   AxisStore[14].Axis[12].Pos13.Position := 0.0;
   AxisStore[14].Axis[12].Pos13.Speed := 0;
   AxisStore[14].Axis[12].Pos13.Reached := FALSE;
   AxisStore[14].Axis[12].Pos14.Position := 0.0;
   AxisStore[14].Axis[12].Pos14.Speed := 0;
   AxisStore[14].Axis[12].Pos14.Reached := FALSE;
   AxisStore[14].Axis[12].Pos15.Position := 0.0;
   AxisStore[14].Axis[12].Pos15.Speed := 0;
   AxisStore[14].Axis[12].Pos15.Reached := FALSE;
   AxisStore[14].Axis[12].Pos16.Position := 0.0;
   AxisStore[14].Axis[12].Pos16.Speed := 0;
   AxisStore[14].Axis[12].Pos16.Reached := FALSE;
   AxisStore[14].Axis[12].Pos17.Position := 0.0;
   AxisStore[14].Axis[12].Pos17.Speed := 0;
   AxisStore[14].Axis[12].Pos17.Reached := FALSE;
   AxisStore[14].Axis[12].Pos18.Position := 0.0;
   AxisStore[14].Axis[12].Pos18.Speed := 0;
   AxisStore[14].Axis[12].Pos18.Reached := FALSE;
   AxisStore[14].Axis[12].Pos19.Position := 0.0;
   AxisStore[14].Axis[12].Pos19.Speed := 0;
   AxisStore[14].Axis[12].Pos19.Reached := FALSE;
   AxisStore[14].Axis[12].Pos20.Position := 0.0;
   AxisStore[14].Axis[12].Pos20.Speed := 0;
   AxisStore[14].Axis[12].Pos20.Reached := FALSE;
   AxisStore[14].Axis[12].Pos21.Position := 0.0;
   AxisStore[14].Axis[12].Pos21.Speed := 0;
   AxisStore[14].Axis[12].Pos21.Reached := FALSE;
   AxisStore[14].Axis[12].Pos22.Position := 0.0;
   AxisStore[14].Axis[12].Pos22.Speed := 0;
   AxisStore[14].Axis[12].Pos22.Reached := FALSE;
   AxisStore[14].Axis[12].Pos23.Position := 0.0;
   AxisStore[14].Axis[12].Pos23.Speed := 0;
   AxisStore[14].Axis[12].Pos23.Reached := FALSE;
   AxisStore[14].Axis[12].Pos24.Position := 0.0;
   AxisStore[14].Axis[12].Pos24.Speed := 0;
   AxisStore[14].Axis[12].Pos24.Reached := FALSE;
   AxisStore[14].Axis[12].Pos25.Position := 0.0;
   AxisStore[14].Axis[12].Pos25.Speed := 0;
   AxisStore[14].Axis[12].Pos25.Reached := FALSE;
   AxisStore[14].Axis[12].Pos26.Position := 0.0;
   AxisStore[14].Axis[12].Pos26.Speed := 0;
   AxisStore[14].Axis[12].Pos26.Reached := FALSE;
   AxisStore[14].Axis[12].Pos27.Position := 0.0;
   AxisStore[14].Axis[12].Pos27.Speed := 0;
   AxisStore[14].Axis[12].Pos27.Reached := FALSE;
   AxisStore[14].Axis[12].Pos28.Position := 0.0;
   AxisStore[14].Axis[12].Pos28.Speed := 0;
   AxisStore[14].Axis[12].Pos28.Reached := FALSE;
   AxisStore[14].Axis[12].Pos29.Position := 0.0;
   AxisStore[14].Axis[12].Pos29.Speed := 0;
   AxisStore[14].Axis[12].Pos29.Reached := FALSE;
   AxisStore[14].Axis[12].Pos30.Position := 0.0;
   AxisStore[14].Axis[12].Pos30.Speed := 0;
   AxisStore[14].Axis[12].Pos30.Reached := FALSE;
   AxisStore[14].Axis[13].Pos1.Position := 0.0;
   AxisStore[14].Axis[13].Pos1.Speed := 0;
   AxisStore[14].Axis[13].Pos1.Reached := FALSE;
   AxisStore[14].Axis[13].Pos2.Position := 0.0;
   AxisStore[14].Axis[13].Pos2.Speed := 0;
   AxisStore[14].Axis[13].Pos2.Reached := FALSE;
   AxisStore[14].Axis[13].Pos3.Position := 0.0;
   AxisStore[14].Axis[13].Pos3.Speed := 0;
   AxisStore[14].Axis[13].Pos3.Reached := FALSE;
   AxisStore[14].Axis[13].Pos4.Position := 0.0;
   AxisStore[14].Axis[13].Pos4.Speed := 0;
   AxisStore[14].Axis[13].Pos4.Reached := FALSE;
   AxisStore[14].Axis[13].Pos5.Position := 0.0;
   AxisStore[14].Axis[13].Pos5.Speed := 0;
   AxisStore[14].Axis[13].Pos5.Reached := FALSE;
   AxisStore[14].Axis[13].Pos6.Position := 0.0;
   AxisStore[14].Axis[13].Pos6.Speed := 0;
   AxisStore[14].Axis[13].Pos6.Reached := FALSE;
   AxisStore[14].Axis[13].Pos7.Position := 0.0;
   AxisStore[14].Axis[13].Pos7.Speed := 0;
   AxisStore[14].Axis[13].Pos7.Reached := FALSE;
   AxisStore[14].Axis[13].Pos8.Position := 0.0;
   AxisStore[14].Axis[13].Pos8.Speed := 0;
   AxisStore[14].Axis[13].Pos8.Reached := FALSE;
   AxisStore[14].Axis[13].Pos9.Position := 0.0;
   AxisStore[14].Axis[13].Pos9.Speed := 0;
   AxisStore[14].Axis[13].Pos9.Reached := FALSE;
   AxisStore[14].Axis[13].Pos10.Position := 0.0;
   AxisStore[14].Axis[13].Pos10.Speed := 0;
   AxisStore[14].Axis[13].Pos10.Reached := FALSE;
   AxisStore[14].Axis[13].Pos11.Position := 0.0;
   AxisStore[14].Axis[13].Pos11.Speed := 0;
   AxisStore[14].Axis[13].Pos11.Reached := FALSE;
   AxisStore[14].Axis[13].Pos12.Position := 0.0;
   AxisStore[14].Axis[13].Pos12.Speed := 0;
   AxisStore[14].Axis[13].Pos12.Reached := FALSE;
   AxisStore[14].Axis[13].Pos13.Position := 0.0;
   AxisStore[14].Axis[13].Pos13.Speed := 0;
   AxisStore[14].Axis[13].Pos13.Reached := FALSE;
   AxisStore[14].Axis[13].Pos14.Position := 0.0;
   AxisStore[14].Axis[13].Pos14.Speed := 0;
   AxisStore[14].Axis[13].Pos14.Reached := FALSE;
   AxisStore[14].Axis[13].Pos15.Position := 0.0;
   AxisStore[14].Axis[13].Pos15.Speed := 0;
   AxisStore[14].Axis[13].Pos15.Reached := FALSE;
   AxisStore[14].Axis[13].Pos16.Position := 0.0;
   AxisStore[14].Axis[13].Pos16.Speed := 0;
   AxisStore[14].Axis[13].Pos16.Reached := FALSE;
   AxisStore[14].Axis[13].Pos17.Position := 0.0;
   AxisStore[14].Axis[13].Pos17.Speed := 0;
   AxisStore[14].Axis[13].Pos17.Reached := FALSE;
   AxisStore[14].Axis[13].Pos18.Position := 0.0;
   AxisStore[14].Axis[13].Pos18.Speed := 0;
   AxisStore[14].Axis[13].Pos18.Reached := FALSE;
   AxisStore[14].Axis[13].Pos19.Position := 0.0;
   AxisStore[14].Axis[13].Pos19.Speed := 0;
   AxisStore[14].Axis[13].Pos19.Reached := FALSE;
   AxisStore[14].Axis[13].Pos20.Position := 0.0;
   AxisStore[14].Axis[13].Pos20.Speed := 0;
   AxisStore[14].Axis[13].Pos20.Reached := FALSE;
   AxisStore[14].Axis[13].Pos21.Position := 0.0;
   AxisStore[14].Axis[13].Pos21.Speed := 0;
   AxisStore[14].Axis[13].Pos21.Reached := FALSE;
   AxisStore[14].Axis[13].Pos22.Position := 0.0;
   AxisStore[14].Axis[13].Pos22.Speed := 0;
   AxisStore[14].Axis[13].Pos22.Reached := FALSE;
   AxisStore[14].Axis[13].Pos23.Position := 0.0;
   AxisStore[14].Axis[13].Pos23.Speed := 0;
   AxisStore[14].Axis[13].Pos23.Reached := FALSE;
   AxisStore[14].Axis[13].Pos24.Position := 0.0;
   AxisStore[14].Axis[13].Pos24.Speed := 0;
   AxisStore[14].Axis[13].Pos24.Reached := FALSE;
   AxisStore[14].Axis[13].Pos25.Position := 0.0;
   AxisStore[14].Axis[13].Pos25.Speed := 0;
   AxisStore[14].Axis[13].Pos25.Reached := FALSE;
   AxisStore[14].Axis[13].Pos26.Position := 0.0;
   AxisStore[14].Axis[13].Pos26.Speed := 0;
   AxisStore[14].Axis[13].Pos26.Reached := FALSE;
   AxisStore[14].Axis[13].Pos27.Position := 0.0;
   AxisStore[14].Axis[13].Pos27.Speed := 0;
   AxisStore[14].Axis[13].Pos27.Reached := FALSE;
   AxisStore[14].Axis[13].Pos28.Position := 0.0;
   AxisStore[14].Axis[13].Pos28.Speed := 0;
   AxisStore[14].Axis[13].Pos28.Reached := FALSE;
   AxisStore[14].Axis[13].Pos29.Position := 0.0;
   AxisStore[14].Axis[13].Pos29.Speed := 0;
   AxisStore[14].Axis[13].Pos29.Reached := FALSE;
   AxisStore[14].Axis[13].Pos30.Position := 0.0;
   AxisStore[14].Axis[13].Pos30.Speed := 0;
   AxisStore[14].Axis[13].Pos30.Reached := FALSE;
   AxisStore[14].Axis[14].Pos1.Position := 0.0;
   AxisStore[14].Axis[14].Pos1.Speed := 0;
   AxisStore[14].Axis[14].Pos1.Reached := FALSE;
   AxisStore[14].Axis[14].Pos2.Position := 0.0;
   AxisStore[14].Axis[14].Pos2.Speed := 0;
   AxisStore[14].Axis[14].Pos2.Reached := FALSE;
   AxisStore[14].Axis[14].Pos3.Position := 0.0;
   AxisStore[14].Axis[14].Pos3.Speed := 0;
   AxisStore[14].Axis[14].Pos3.Reached := FALSE;
   AxisStore[14].Axis[14].Pos4.Position := 0.0;
   AxisStore[14].Axis[14].Pos4.Speed := 0;
   AxisStore[14].Axis[14].Pos4.Reached := FALSE;
   AxisStore[14].Axis[14].Pos5.Position := 0.0;
   AxisStore[14].Axis[14].Pos5.Speed := 0;
   AxisStore[14].Axis[14].Pos5.Reached := FALSE;
   AxisStore[14].Axis[14].Pos6.Position := 0.0;
   AxisStore[14].Axis[14].Pos6.Speed := 0;
   AxisStore[14].Axis[14].Pos6.Reached := FALSE;
   AxisStore[14].Axis[14].Pos7.Position := 0.0;
   AxisStore[14].Axis[14].Pos7.Speed := 0;
   AxisStore[14].Axis[14].Pos7.Reached := FALSE;
   AxisStore[14].Axis[14].Pos8.Position := 0.0;
   AxisStore[14].Axis[14].Pos8.Speed := 0;
   AxisStore[14].Axis[14].Pos8.Reached := FALSE;
   AxisStore[14].Axis[14].Pos9.Position := 0.0;
   AxisStore[14].Axis[14].Pos9.Speed := 0;
   AxisStore[14].Axis[14].Pos9.Reached := FALSE;
   AxisStore[14].Axis[14].Pos10.Position := 0.0;
   AxisStore[14].Axis[14].Pos10.Speed := 0;
   AxisStore[14].Axis[14].Pos10.Reached := FALSE;
   AxisStore[14].Axis[14].Pos11.Position := 0.0;
   AxisStore[14].Axis[14].Pos11.Speed := 0;
   AxisStore[14].Axis[14].Pos11.Reached := FALSE;
   AxisStore[14].Axis[14].Pos12.Position := 0.0;
   AxisStore[14].Axis[14].Pos12.Speed := 0;
   AxisStore[14].Axis[14].Pos12.Reached := FALSE;
   AxisStore[14].Axis[14].Pos13.Position := 0.0;
   AxisStore[14].Axis[14].Pos13.Speed := 0;
   AxisStore[14].Axis[14].Pos13.Reached := FALSE;
   AxisStore[14].Axis[14].Pos14.Position := 0.0;
   AxisStore[14].Axis[14].Pos14.Speed := 0;
   AxisStore[14].Axis[14].Pos14.Reached := FALSE;
   AxisStore[14].Axis[14].Pos15.Position := 0.0;
   AxisStore[14].Axis[14].Pos15.Speed := 0;
   AxisStore[14].Axis[14].Pos15.Reached := FALSE;
   AxisStore[14].Axis[14].Pos16.Position := 0.0;
   AxisStore[14].Axis[14].Pos16.Speed := 0;
   AxisStore[14].Axis[14].Pos16.Reached := FALSE;
   AxisStore[14].Axis[14].Pos17.Position := 0.0;
   AxisStore[14].Axis[14].Pos17.Speed := 0;
   AxisStore[14].Axis[14].Pos17.Reached := FALSE;
   AxisStore[14].Axis[14].Pos18.Position := 0.0;
   AxisStore[14].Axis[14].Pos18.Speed := 0;
   AxisStore[14].Axis[14].Pos18.Reached := FALSE;
   AxisStore[14].Axis[14].Pos19.Position := 0.0;
   AxisStore[14].Axis[14].Pos19.Speed := 0;
   AxisStore[14].Axis[14].Pos19.Reached := FALSE;
   AxisStore[14].Axis[14].Pos20.Position := 0.0;
   AxisStore[14].Axis[14].Pos20.Speed := 0;
   AxisStore[14].Axis[14].Pos20.Reached := FALSE;
   AxisStore[14].Axis[14].Pos21.Position := 0.0;
   AxisStore[14].Axis[14].Pos21.Speed := 0;
   AxisStore[14].Axis[14].Pos21.Reached := FALSE;
   AxisStore[14].Axis[14].Pos22.Position := 0.0;
   AxisStore[14].Axis[14].Pos22.Speed := 0;
   AxisStore[14].Axis[14].Pos22.Reached := FALSE;
   AxisStore[14].Axis[14].Pos23.Position := 0.0;
   AxisStore[14].Axis[14].Pos23.Speed := 0;
   AxisStore[14].Axis[14].Pos23.Reached := FALSE;
   AxisStore[14].Axis[14].Pos24.Position := 0.0;
   AxisStore[14].Axis[14].Pos24.Speed := 0;
   AxisStore[14].Axis[14].Pos24.Reached := FALSE;
   AxisStore[14].Axis[14].Pos25.Position := 0.0;
   AxisStore[14].Axis[14].Pos25.Speed := 0;
   AxisStore[14].Axis[14].Pos25.Reached := FALSE;
   AxisStore[14].Axis[14].Pos26.Position := 0.0;
   AxisStore[14].Axis[14].Pos26.Speed := 0;
   AxisStore[14].Axis[14].Pos26.Reached := FALSE;
   AxisStore[14].Axis[14].Pos27.Position := 0.0;
   AxisStore[14].Axis[14].Pos27.Speed := 0;
   AxisStore[14].Axis[14].Pos27.Reached := FALSE;
   AxisStore[14].Axis[14].Pos28.Position := 0.0;
   AxisStore[14].Axis[14].Pos28.Speed := 0;
   AxisStore[14].Axis[14].Pos28.Reached := FALSE;
   AxisStore[14].Axis[14].Pos29.Position := 0.0;
   AxisStore[14].Axis[14].Pos29.Speed := 0;
   AxisStore[14].Axis[14].Pos29.Reached := FALSE;
   AxisStore[14].Axis[14].Pos30.Position := 0.0;
   AxisStore[14].Axis[14].Pos30.Speed := 0;
   AxisStore[14].Axis[14].Pos30.Reached := FALSE;
   AxisStore[14].Axis[15].Pos1.Position := 0.0;
   AxisStore[14].Axis[15].Pos1.Speed := 0;
   AxisStore[14].Axis[15].Pos1.Reached := FALSE;
   AxisStore[14].Axis[15].Pos2.Position := 0.0;
   AxisStore[14].Axis[15].Pos2.Speed := 0;
   AxisStore[14].Axis[15].Pos2.Reached := FALSE;
   AxisStore[14].Axis[15].Pos3.Position := 0.0;
   AxisStore[14].Axis[15].Pos3.Speed := 0;
   AxisStore[14].Axis[15].Pos3.Reached := FALSE;
   AxisStore[14].Axis[15].Pos4.Position := 0.0;
   AxisStore[14].Axis[15].Pos4.Speed := 0;
   AxisStore[14].Axis[15].Pos4.Reached := FALSE;
   AxisStore[14].Axis[15].Pos5.Position := 0.0;
   AxisStore[14].Axis[15].Pos5.Speed := 0;
   AxisStore[14].Axis[15].Pos5.Reached := FALSE;
   AxisStore[14].Axis[15].Pos6.Position := 0.0;
   AxisStore[14].Axis[15].Pos6.Speed := 0;
   AxisStore[14].Axis[15].Pos6.Reached := FALSE;
   AxisStore[14].Axis[15].Pos7.Position := 0.0;
   AxisStore[14].Axis[15].Pos7.Speed := 0;
   AxisStore[14].Axis[15].Pos7.Reached := FALSE;
   AxisStore[14].Axis[15].Pos8.Position := 0.0;
   AxisStore[14].Axis[15].Pos8.Speed := 0;
   AxisStore[14].Axis[15].Pos8.Reached := FALSE;
   AxisStore[14].Axis[15].Pos9.Position := 0.0;
   AxisStore[14].Axis[15].Pos9.Speed := 0;
   AxisStore[14].Axis[15].Pos9.Reached := FALSE;
   AxisStore[14].Axis[15].Pos10.Position := 0.0;
   AxisStore[14].Axis[15].Pos10.Speed := 0;
   AxisStore[14].Axis[15].Pos10.Reached := FALSE;
   AxisStore[14].Axis[15].Pos11.Position := 0.0;
   AxisStore[14].Axis[15].Pos11.Speed := 0;
   AxisStore[14].Axis[15].Pos11.Reached := FALSE;
   AxisStore[14].Axis[15].Pos12.Position := 0.0;
   AxisStore[14].Axis[15].Pos12.Speed := 0;
   AxisStore[14].Axis[15].Pos12.Reached := FALSE;
   AxisStore[14].Axis[15].Pos13.Position := 0.0;
   AxisStore[14].Axis[15].Pos13.Speed := 0;
   AxisStore[14].Axis[15].Pos13.Reached := FALSE;
   AxisStore[14].Axis[15].Pos14.Position := 0.0;
   AxisStore[14].Axis[15].Pos14.Speed := 0;
   AxisStore[14].Axis[15].Pos14.Reached := FALSE;
   AxisStore[14].Axis[15].Pos15.Position := 0.0;
   AxisStore[14].Axis[15].Pos15.Speed := 0;
   AxisStore[14].Axis[15].Pos15.Reached := FALSE;
   AxisStore[14].Axis[15].Pos16.Position := 0.0;
   AxisStore[14].Axis[15].Pos16.Speed := 0;
   AxisStore[14].Axis[15].Pos16.Reached := FALSE;
   AxisStore[14].Axis[15].Pos17.Position := 0.0;
   AxisStore[14].Axis[15].Pos17.Speed := 0;
   AxisStore[14].Axis[15].Pos17.Reached := FALSE;
   AxisStore[14].Axis[15].Pos18.Position := 0.0;
   AxisStore[14].Axis[15].Pos18.Speed := 0;
   AxisStore[14].Axis[15].Pos18.Reached := FALSE;
   AxisStore[14].Axis[15].Pos19.Position := 0.0;
   AxisStore[14].Axis[15].Pos19.Speed := 0;
   AxisStore[14].Axis[15].Pos19.Reached := FALSE;
   AxisStore[14].Axis[15].Pos20.Position := 0.0;
   AxisStore[14].Axis[15].Pos20.Speed := 0;
   AxisStore[14].Axis[15].Pos20.Reached := FALSE;
   AxisStore[14].Axis[15].Pos21.Position := 0.0;
   AxisStore[14].Axis[15].Pos21.Speed := 0;
   AxisStore[14].Axis[15].Pos21.Reached := FALSE;
   AxisStore[14].Axis[15].Pos22.Position := 0.0;
   AxisStore[14].Axis[15].Pos22.Speed := 0;
   AxisStore[14].Axis[15].Pos22.Reached := FALSE;
   AxisStore[14].Axis[15].Pos23.Position := 0.0;
   AxisStore[14].Axis[15].Pos23.Speed := 0;
   AxisStore[14].Axis[15].Pos23.Reached := FALSE;
   AxisStore[14].Axis[15].Pos24.Position := 0.0;
   AxisStore[14].Axis[15].Pos24.Speed := 0;
   AxisStore[14].Axis[15].Pos24.Reached := FALSE;
   AxisStore[14].Axis[15].Pos25.Position := 0.0;
   AxisStore[14].Axis[15].Pos25.Speed := 0;
   AxisStore[14].Axis[15].Pos25.Reached := FALSE;
   AxisStore[14].Axis[15].Pos26.Position := 0.0;
   AxisStore[14].Axis[15].Pos26.Speed := 0;
   AxisStore[14].Axis[15].Pos26.Reached := FALSE;
   AxisStore[14].Axis[15].Pos27.Position := 0.0;
   AxisStore[14].Axis[15].Pos27.Speed := 0;
   AxisStore[14].Axis[15].Pos27.Reached := FALSE;
   AxisStore[14].Axis[15].Pos28.Position := 0.0;
   AxisStore[14].Axis[15].Pos28.Speed := 0;
   AxisStore[14].Axis[15].Pos28.Reached := FALSE;
   AxisStore[14].Axis[15].Pos29.Position := 0.0;
   AxisStore[14].Axis[15].Pos29.Speed := 0;
   AxisStore[14].Axis[15].Pos29.Reached := FALSE;
   AxisStore[14].Axis[15].Pos30.Position := 0.0;
   AxisStore[14].Axis[15].Pos30.Speed := 0;
   AxisStore[14].Axis[15].Pos30.Reached := FALSE;
   AxisStore[15].Axis[1].Pos1.Position := 0.0;
   AxisStore[15].Axis[1].Pos1.Speed := 0;
   AxisStore[15].Axis[1].Pos1.Reached := FALSE;
   AxisStore[15].Axis[1].Pos2.Position := 0.0;
   AxisStore[15].Axis[1].Pos2.Speed := 0;
   AxisStore[15].Axis[1].Pos2.Reached := FALSE;
   AxisStore[15].Axis[1].Pos3.Position := 0.0;
   AxisStore[15].Axis[1].Pos3.Speed := 0;
   AxisStore[15].Axis[1].Pos3.Reached := FALSE;
   AxisStore[15].Axis[1].Pos4.Position := 0.0;
   AxisStore[15].Axis[1].Pos4.Speed := 0;
   AxisStore[15].Axis[1].Pos4.Reached := FALSE;
   AxisStore[15].Axis[1].Pos5.Position := 0.0;
   AxisStore[15].Axis[1].Pos5.Speed := 0;
   AxisStore[15].Axis[1].Pos5.Reached := FALSE;
   AxisStore[15].Axis[1].Pos6.Position := 0.0;
   AxisStore[15].Axis[1].Pos6.Speed := 0;
   AxisStore[15].Axis[1].Pos6.Reached := FALSE;
   AxisStore[15].Axis[1].Pos7.Position := 0.0;
   AxisStore[15].Axis[1].Pos7.Speed := 0;
   AxisStore[15].Axis[1].Pos7.Reached := FALSE;
   AxisStore[15].Axis[1].Pos8.Position := 0.0;
   AxisStore[15].Axis[1].Pos8.Speed := 0;
   AxisStore[15].Axis[1].Pos8.Reached := FALSE;
   AxisStore[15].Axis[1].Pos9.Position := 0.0;
   AxisStore[15].Axis[1].Pos9.Speed := 0;
   AxisStore[15].Axis[1].Pos9.Reached := FALSE;
   AxisStore[15].Axis[1].Pos10.Position := 0.0;
   AxisStore[15].Axis[1].Pos10.Speed := 0;
   AxisStore[15].Axis[1].Pos10.Reached := FALSE;
   AxisStore[15].Axis[1].Pos11.Position := 0.0;
   AxisStore[15].Axis[1].Pos11.Speed := 0;
   AxisStore[15].Axis[1].Pos11.Reached := FALSE;
   AxisStore[15].Axis[1].Pos12.Position := 0.0;
   AxisStore[15].Axis[1].Pos12.Speed := 0;
   AxisStore[15].Axis[1].Pos12.Reached := FALSE;
   AxisStore[15].Axis[1].Pos13.Position := 0.0;
   AxisStore[15].Axis[1].Pos13.Speed := 0;
   AxisStore[15].Axis[1].Pos13.Reached := FALSE;
   AxisStore[15].Axis[1].Pos14.Position := 0.0;
   AxisStore[15].Axis[1].Pos14.Speed := 0;
   AxisStore[15].Axis[1].Pos14.Reached := FALSE;
   AxisStore[15].Axis[1].Pos15.Position := 0.0;
   AxisStore[15].Axis[1].Pos15.Speed := 0;
   AxisStore[15].Axis[1].Pos15.Reached := FALSE;
   AxisStore[15].Axis[1].Pos16.Position := 0.0;
   AxisStore[15].Axis[1].Pos16.Speed := 0;
   AxisStore[15].Axis[1].Pos16.Reached := FALSE;
   AxisStore[15].Axis[1].Pos17.Position := 0.0;
   AxisStore[15].Axis[1].Pos17.Speed := 0;
   AxisStore[15].Axis[1].Pos17.Reached := FALSE;
   AxisStore[15].Axis[1].Pos18.Position := 0.0;
   AxisStore[15].Axis[1].Pos18.Speed := 0;
   AxisStore[15].Axis[1].Pos18.Reached := FALSE;
   AxisStore[15].Axis[1].Pos19.Position := 0.0;
   AxisStore[15].Axis[1].Pos19.Speed := 0;
   AxisStore[15].Axis[1].Pos19.Reached := FALSE;
   AxisStore[15].Axis[1].Pos20.Position := 0.0;
   AxisStore[15].Axis[1].Pos20.Speed := 0;
   AxisStore[15].Axis[1].Pos20.Reached := FALSE;
   AxisStore[15].Axis[1].Pos21.Position := 0.0;
   AxisStore[15].Axis[1].Pos21.Speed := 0;
   AxisStore[15].Axis[1].Pos21.Reached := FALSE;
   AxisStore[15].Axis[1].Pos22.Position := 0.0;
   AxisStore[15].Axis[1].Pos22.Speed := 0;
   AxisStore[15].Axis[1].Pos22.Reached := FALSE;
   AxisStore[15].Axis[1].Pos23.Position := 0.0;
   AxisStore[15].Axis[1].Pos23.Speed := 0;
   AxisStore[15].Axis[1].Pos23.Reached := FALSE;
   AxisStore[15].Axis[1].Pos24.Position := 0.0;
   AxisStore[15].Axis[1].Pos24.Speed := 0;
   AxisStore[15].Axis[1].Pos24.Reached := FALSE;
   AxisStore[15].Axis[1].Pos25.Position := 0.0;
   AxisStore[15].Axis[1].Pos25.Speed := 0;
   AxisStore[15].Axis[1].Pos25.Reached := FALSE;
   AxisStore[15].Axis[1].Pos26.Position := 0.0;
   AxisStore[15].Axis[1].Pos26.Speed := 0;
   AxisStore[15].Axis[1].Pos26.Reached := FALSE;
   AxisStore[15].Axis[1].Pos27.Position := 0.0;
   AxisStore[15].Axis[1].Pos27.Speed := 0;
   AxisStore[15].Axis[1].Pos27.Reached := FALSE;
   AxisStore[15].Axis[1].Pos28.Position := 0.0;
   AxisStore[15].Axis[1].Pos28.Speed := 0;
   AxisStore[15].Axis[1].Pos28.Reached := FALSE;
   AxisStore[15].Axis[1].Pos29.Position := 0.0;
   AxisStore[15].Axis[1].Pos29.Speed := 0;
   AxisStore[15].Axis[1].Pos29.Reached := FALSE;
   AxisStore[15].Axis[1].Pos30.Position := 0.0;
   AxisStore[15].Axis[1].Pos30.Speed := 0;
   AxisStore[15].Axis[1].Pos30.Reached := FALSE;
   AxisStore[15].Axis[2].Pos1.Position := 0.0;
   AxisStore[15].Axis[2].Pos1.Speed := 0;
   AxisStore[15].Axis[2].Pos1.Reached := FALSE;
   AxisStore[15].Axis[2].Pos2.Position := 0.0;
   AxisStore[15].Axis[2].Pos2.Speed := 0;
   AxisStore[15].Axis[2].Pos2.Reached := FALSE;
   AxisStore[15].Axis[2].Pos3.Position := 0.0;
   AxisStore[15].Axis[2].Pos3.Speed := 0;
   AxisStore[15].Axis[2].Pos3.Reached := FALSE;
   AxisStore[15].Axis[2].Pos4.Position := 0.0;
   AxisStore[15].Axis[2].Pos4.Speed := 0;
   AxisStore[15].Axis[2].Pos4.Reached := FALSE;
   AxisStore[15].Axis[2].Pos5.Position := 0.0;
   AxisStore[15].Axis[2].Pos5.Speed := 0;
   AxisStore[15].Axis[2].Pos5.Reached := FALSE;
   AxisStore[15].Axis[2].Pos6.Position := 0.0;
   AxisStore[15].Axis[2].Pos6.Speed := 0;
   AxisStore[15].Axis[2].Pos6.Reached := FALSE;
   AxisStore[15].Axis[2].Pos7.Position := 0.0;
   AxisStore[15].Axis[2].Pos7.Speed := 0;
   AxisStore[15].Axis[2].Pos7.Reached := FALSE;
   AxisStore[15].Axis[2].Pos8.Position := 0.0;
   AxisStore[15].Axis[2].Pos8.Speed := 0;
   AxisStore[15].Axis[2].Pos8.Reached := FALSE;
   AxisStore[15].Axis[2].Pos9.Position := 0.0;
   AxisStore[15].Axis[2].Pos9.Speed := 0;
   AxisStore[15].Axis[2].Pos9.Reached := FALSE;
   AxisStore[15].Axis[2].Pos10.Position := 0.0;
   AxisStore[15].Axis[2].Pos10.Speed := 0;
   AxisStore[15].Axis[2].Pos10.Reached := FALSE;
   AxisStore[15].Axis[2].Pos11.Position := 0.0;
   AxisStore[15].Axis[2].Pos11.Speed := 0;
   AxisStore[15].Axis[2].Pos11.Reached := FALSE;
   AxisStore[15].Axis[2].Pos12.Position := 0.0;
   AxisStore[15].Axis[2].Pos12.Speed := 0;
   AxisStore[15].Axis[2].Pos12.Reached := FALSE;
   AxisStore[15].Axis[2].Pos13.Position := 0.0;
   AxisStore[15].Axis[2].Pos13.Speed := 0;
   AxisStore[15].Axis[2].Pos13.Reached := FALSE;
   AxisStore[15].Axis[2].Pos14.Position := 0.0;
   AxisStore[15].Axis[2].Pos14.Speed := 0;
   AxisStore[15].Axis[2].Pos14.Reached := FALSE;
   AxisStore[15].Axis[2].Pos15.Position := 0.0;
   AxisStore[15].Axis[2].Pos15.Speed := 0;
   AxisStore[15].Axis[2].Pos15.Reached := FALSE;
   AxisStore[15].Axis[2].Pos16.Position := 0.0;
   AxisStore[15].Axis[2].Pos16.Speed := 0;
   AxisStore[15].Axis[2].Pos16.Reached := FALSE;
   AxisStore[15].Axis[2].Pos17.Position := 0.0;
   AxisStore[15].Axis[2].Pos17.Speed := 0;
   AxisStore[15].Axis[2].Pos17.Reached := FALSE;
   AxisStore[15].Axis[2].Pos18.Position := 0.0;
   AxisStore[15].Axis[2].Pos18.Speed := 0;
   AxisStore[15].Axis[2].Pos18.Reached := FALSE;
   AxisStore[15].Axis[2].Pos19.Position := 0.0;
   AxisStore[15].Axis[2].Pos19.Speed := 0;
   AxisStore[15].Axis[2].Pos19.Reached := FALSE;
   AxisStore[15].Axis[2].Pos20.Position := 0.0;
   AxisStore[15].Axis[2].Pos20.Speed := 0;
   AxisStore[15].Axis[2].Pos20.Reached := FALSE;
   AxisStore[15].Axis[2].Pos21.Position := 0.0;
   AxisStore[15].Axis[2].Pos21.Speed := 0;
   AxisStore[15].Axis[2].Pos21.Reached := FALSE;
   AxisStore[15].Axis[2].Pos22.Position := 0.0;
   AxisStore[15].Axis[2].Pos22.Speed := 0;
   AxisStore[15].Axis[2].Pos22.Reached := FALSE;
   AxisStore[15].Axis[2].Pos23.Position := 0.0;
   AxisStore[15].Axis[2].Pos23.Speed := 0;
   AxisStore[15].Axis[2].Pos23.Reached := FALSE;
   AxisStore[15].Axis[2].Pos24.Position := 0.0;
   AxisStore[15].Axis[2].Pos24.Speed := 0;
   AxisStore[15].Axis[2].Pos24.Reached := FALSE;
   AxisStore[15].Axis[2].Pos25.Position := 0.0;
   AxisStore[15].Axis[2].Pos25.Speed := 0;
   AxisStore[15].Axis[2].Pos25.Reached := FALSE;
   AxisStore[15].Axis[2].Pos26.Position := 0.0;
   AxisStore[15].Axis[2].Pos26.Speed := 0;
   AxisStore[15].Axis[2].Pos26.Reached := FALSE;
   AxisStore[15].Axis[2].Pos27.Position := 0.0;
   AxisStore[15].Axis[2].Pos27.Speed := 0;
   AxisStore[15].Axis[2].Pos27.Reached := FALSE;
   AxisStore[15].Axis[2].Pos28.Position := 0.0;
   AxisStore[15].Axis[2].Pos28.Speed := 0;
   AxisStore[15].Axis[2].Pos28.Reached := FALSE;
   AxisStore[15].Axis[2].Pos29.Position := 0.0;
   AxisStore[15].Axis[2].Pos29.Speed := 0;
   AxisStore[15].Axis[2].Pos29.Reached := FALSE;
   AxisStore[15].Axis[2].Pos30.Position := 0.0;
   AxisStore[15].Axis[2].Pos30.Speed := 0;
   AxisStore[15].Axis[2].Pos30.Reached := FALSE;
   AxisStore[15].Axis[3].Pos1.Position := 0.0;
   AxisStore[15].Axis[3].Pos1.Speed := 0;
   AxisStore[15].Axis[3].Pos1.Reached := FALSE;
   AxisStore[15].Axis[3].Pos2.Position := 0.0;
   AxisStore[15].Axis[3].Pos2.Speed := 0;
   AxisStore[15].Axis[3].Pos2.Reached := FALSE;
   AxisStore[15].Axis[3].Pos3.Position := 0.0;
   AxisStore[15].Axis[3].Pos3.Speed := 0;
   AxisStore[15].Axis[3].Pos3.Reached := FALSE;
   AxisStore[15].Axis[3].Pos4.Position := 0.0;
   AxisStore[15].Axis[3].Pos4.Speed := 0;
   AxisStore[15].Axis[3].Pos4.Reached := FALSE;
   AxisStore[15].Axis[3].Pos5.Position := 0.0;
   AxisStore[15].Axis[3].Pos5.Speed := 0;
   AxisStore[15].Axis[3].Pos5.Reached := FALSE;
   AxisStore[15].Axis[3].Pos6.Position := 0.0;
   AxisStore[15].Axis[3].Pos6.Speed := 0;
   AxisStore[15].Axis[3].Pos6.Reached := FALSE;
   AxisStore[15].Axis[3].Pos7.Position := 0.0;
   AxisStore[15].Axis[3].Pos7.Speed := 0;
   AxisStore[15].Axis[3].Pos7.Reached := FALSE;
   AxisStore[15].Axis[3].Pos8.Position := 0.0;
   AxisStore[15].Axis[3].Pos8.Speed := 0;
   AxisStore[15].Axis[3].Pos8.Reached := FALSE;
   AxisStore[15].Axis[3].Pos9.Position := 0.0;
   AxisStore[15].Axis[3].Pos9.Speed := 0;
   AxisStore[15].Axis[3].Pos9.Reached := FALSE;
   AxisStore[15].Axis[3].Pos10.Position := 0.0;
   AxisStore[15].Axis[3].Pos10.Speed := 0;
   AxisStore[15].Axis[3].Pos10.Reached := FALSE;
   AxisStore[15].Axis[3].Pos11.Position := 0.0;
   AxisStore[15].Axis[3].Pos11.Speed := 0;
   AxisStore[15].Axis[3].Pos11.Reached := FALSE;
   AxisStore[15].Axis[3].Pos12.Position := 0.0;
   AxisStore[15].Axis[3].Pos12.Speed := 0;
   AxisStore[15].Axis[3].Pos12.Reached := FALSE;
   AxisStore[15].Axis[3].Pos13.Position := 0.0;
   AxisStore[15].Axis[3].Pos13.Speed := 0;
   AxisStore[15].Axis[3].Pos13.Reached := FALSE;
   AxisStore[15].Axis[3].Pos14.Position := 0.0;
   AxisStore[15].Axis[3].Pos14.Speed := 0;
   AxisStore[15].Axis[3].Pos14.Reached := FALSE;
   AxisStore[15].Axis[3].Pos15.Position := 0.0;
   AxisStore[15].Axis[3].Pos15.Speed := 0;
   AxisStore[15].Axis[3].Pos15.Reached := FALSE;
   AxisStore[15].Axis[3].Pos16.Position := 0.0;
   AxisStore[15].Axis[3].Pos16.Speed := 0;
   AxisStore[15].Axis[3].Pos16.Reached := FALSE;
   AxisStore[15].Axis[3].Pos17.Position := 0.0;
   AxisStore[15].Axis[3].Pos17.Speed := 0;
   AxisStore[15].Axis[3].Pos17.Reached := FALSE;
   AxisStore[15].Axis[3].Pos18.Position := 0.0;
   AxisStore[15].Axis[3].Pos18.Speed := 0;
   AxisStore[15].Axis[3].Pos18.Reached := FALSE;
   AxisStore[15].Axis[3].Pos19.Position := 0.0;
   AxisStore[15].Axis[3].Pos19.Speed := 0;
   AxisStore[15].Axis[3].Pos19.Reached := FALSE;
   AxisStore[15].Axis[3].Pos20.Position := 0.0;
   AxisStore[15].Axis[3].Pos20.Speed := 0;
   AxisStore[15].Axis[3].Pos20.Reached := FALSE;
   AxisStore[15].Axis[3].Pos21.Position := 0.0;
   AxisStore[15].Axis[3].Pos21.Speed := 0;
   AxisStore[15].Axis[3].Pos21.Reached := FALSE;
   AxisStore[15].Axis[3].Pos22.Position := 0.0;
   AxisStore[15].Axis[3].Pos22.Speed := 0;
   AxisStore[15].Axis[3].Pos22.Reached := FALSE;
   AxisStore[15].Axis[3].Pos23.Position := 0.0;
   AxisStore[15].Axis[3].Pos23.Speed := 0;
   AxisStore[15].Axis[3].Pos23.Reached := FALSE;
   AxisStore[15].Axis[3].Pos24.Position := 0.0;
   AxisStore[15].Axis[3].Pos24.Speed := 0;
   AxisStore[15].Axis[3].Pos24.Reached := FALSE;
   AxisStore[15].Axis[3].Pos25.Position := 0.0;
   AxisStore[15].Axis[3].Pos25.Speed := 0;
   AxisStore[15].Axis[3].Pos25.Reached := FALSE;
   AxisStore[15].Axis[3].Pos26.Position := 0.0;
   AxisStore[15].Axis[3].Pos26.Speed := 0;
   AxisStore[15].Axis[3].Pos26.Reached := FALSE;
   AxisStore[15].Axis[3].Pos27.Position := 0.0;
   AxisStore[15].Axis[3].Pos27.Speed := 0;
   AxisStore[15].Axis[3].Pos27.Reached := FALSE;
   AxisStore[15].Axis[3].Pos28.Position := 0.0;
   AxisStore[15].Axis[3].Pos28.Speed := 0;
   AxisStore[15].Axis[3].Pos28.Reached := FALSE;
   AxisStore[15].Axis[3].Pos29.Position := 0.0;
   AxisStore[15].Axis[3].Pos29.Speed := 0;
   AxisStore[15].Axis[3].Pos29.Reached := FALSE;
   AxisStore[15].Axis[3].Pos30.Position := 0.0;
   AxisStore[15].Axis[3].Pos30.Speed := 0;
   AxisStore[15].Axis[3].Pos30.Reached := FALSE;
   AxisStore[15].Axis[4].Pos1.Position := 0.0;
   AxisStore[15].Axis[4].Pos1.Speed := 0;
   AxisStore[15].Axis[4].Pos1.Reached := FALSE;
   AxisStore[15].Axis[4].Pos2.Position := 0.0;
   AxisStore[15].Axis[4].Pos2.Speed := 0;
   AxisStore[15].Axis[4].Pos2.Reached := FALSE;
   AxisStore[15].Axis[4].Pos3.Position := 0.0;
   AxisStore[15].Axis[4].Pos3.Speed := 0;
   AxisStore[15].Axis[4].Pos3.Reached := FALSE;
   AxisStore[15].Axis[4].Pos4.Position := 0.0;
   AxisStore[15].Axis[4].Pos4.Speed := 0;
   AxisStore[15].Axis[4].Pos4.Reached := FALSE;
   AxisStore[15].Axis[4].Pos5.Position := 0.0;
   AxisStore[15].Axis[4].Pos5.Speed := 0;
   AxisStore[15].Axis[4].Pos5.Reached := FALSE;
   AxisStore[15].Axis[4].Pos6.Position := 0.0;
   AxisStore[15].Axis[4].Pos6.Speed := 0;
   AxisStore[15].Axis[4].Pos6.Reached := FALSE;
   AxisStore[15].Axis[4].Pos7.Position := 0.0;
   AxisStore[15].Axis[4].Pos7.Speed := 0;
   AxisStore[15].Axis[4].Pos7.Reached := FALSE;
   AxisStore[15].Axis[4].Pos8.Position := 0.0;
   AxisStore[15].Axis[4].Pos8.Speed := 0;
   AxisStore[15].Axis[4].Pos8.Reached := FALSE;
   AxisStore[15].Axis[4].Pos9.Position := 0.0;
   AxisStore[15].Axis[4].Pos9.Speed := 0;
   AxisStore[15].Axis[4].Pos9.Reached := FALSE;
   AxisStore[15].Axis[4].Pos10.Position := 0.0;
   AxisStore[15].Axis[4].Pos10.Speed := 0;
   AxisStore[15].Axis[4].Pos10.Reached := FALSE;
   AxisStore[15].Axis[4].Pos11.Position := 0.0;
   AxisStore[15].Axis[4].Pos11.Speed := 0;
   AxisStore[15].Axis[4].Pos11.Reached := FALSE;
   AxisStore[15].Axis[4].Pos12.Position := 0.0;
   AxisStore[15].Axis[4].Pos12.Speed := 0;
   AxisStore[15].Axis[4].Pos12.Reached := FALSE;
   AxisStore[15].Axis[4].Pos13.Position := 0.0;
   AxisStore[15].Axis[4].Pos13.Speed := 0;
   AxisStore[15].Axis[4].Pos13.Reached := FALSE;
   AxisStore[15].Axis[4].Pos14.Position := 0.0;
   AxisStore[15].Axis[4].Pos14.Speed := 0;
   AxisStore[15].Axis[4].Pos14.Reached := FALSE;
   AxisStore[15].Axis[4].Pos15.Position := 0.0;
   AxisStore[15].Axis[4].Pos15.Speed := 0;
   AxisStore[15].Axis[4].Pos15.Reached := FALSE;
   AxisStore[15].Axis[4].Pos16.Position := 0.0;
   AxisStore[15].Axis[4].Pos16.Speed := 0;
   AxisStore[15].Axis[4].Pos16.Reached := FALSE;
   AxisStore[15].Axis[4].Pos17.Position := 0.0;
   AxisStore[15].Axis[4].Pos17.Speed := 0;
   AxisStore[15].Axis[4].Pos17.Reached := FALSE;
   AxisStore[15].Axis[4].Pos18.Position := 0.0;
   AxisStore[15].Axis[4].Pos18.Speed := 0;
   AxisStore[15].Axis[4].Pos18.Reached := FALSE;
   AxisStore[15].Axis[4].Pos19.Position := 0.0;
   AxisStore[15].Axis[4].Pos19.Speed := 0;
   AxisStore[15].Axis[4].Pos19.Reached := FALSE;
   AxisStore[15].Axis[4].Pos20.Position := 0.0;
   AxisStore[15].Axis[4].Pos20.Speed := 0;
   AxisStore[15].Axis[4].Pos20.Reached := FALSE;
   AxisStore[15].Axis[4].Pos21.Position := 0.0;
   AxisStore[15].Axis[4].Pos21.Speed := 0;
   AxisStore[15].Axis[4].Pos21.Reached := FALSE;
   AxisStore[15].Axis[4].Pos22.Position := 0.0;
   AxisStore[15].Axis[4].Pos22.Speed := 0;
   AxisStore[15].Axis[4].Pos22.Reached := FALSE;
   AxisStore[15].Axis[4].Pos23.Position := 0.0;
   AxisStore[15].Axis[4].Pos23.Speed := 0;
   AxisStore[15].Axis[4].Pos23.Reached := FALSE;
   AxisStore[15].Axis[4].Pos24.Position := 0.0;
   AxisStore[15].Axis[4].Pos24.Speed := 0;
   AxisStore[15].Axis[4].Pos24.Reached := FALSE;
   AxisStore[15].Axis[4].Pos25.Position := 0.0;
   AxisStore[15].Axis[4].Pos25.Speed := 0;
   AxisStore[15].Axis[4].Pos25.Reached := FALSE;
   AxisStore[15].Axis[4].Pos26.Position := 0.0;
   AxisStore[15].Axis[4].Pos26.Speed := 0;
   AxisStore[15].Axis[4].Pos26.Reached := FALSE;
   AxisStore[15].Axis[4].Pos27.Position := 0.0;
   AxisStore[15].Axis[4].Pos27.Speed := 0;
   AxisStore[15].Axis[4].Pos27.Reached := FALSE;
   AxisStore[15].Axis[4].Pos28.Position := 0.0;
   AxisStore[15].Axis[4].Pos28.Speed := 0;
   AxisStore[15].Axis[4].Pos28.Reached := FALSE;
   AxisStore[15].Axis[4].Pos29.Position := 0.0;
   AxisStore[15].Axis[4].Pos29.Speed := 0;
   AxisStore[15].Axis[4].Pos29.Reached := FALSE;
   AxisStore[15].Axis[4].Pos30.Position := 0.0;
   AxisStore[15].Axis[4].Pos30.Speed := 0;
   AxisStore[15].Axis[4].Pos30.Reached := FALSE;
   AxisStore[15].Axis[5].Pos1.Position := 0.0;
   AxisStore[15].Axis[5].Pos1.Speed := 0;
   AxisStore[15].Axis[5].Pos1.Reached := FALSE;
   AxisStore[15].Axis[5].Pos2.Position := 0.0;
   AxisStore[15].Axis[5].Pos2.Speed := 0;
   AxisStore[15].Axis[5].Pos2.Reached := FALSE;
   AxisStore[15].Axis[5].Pos3.Position := 0.0;
   AxisStore[15].Axis[5].Pos3.Speed := 0;
   AxisStore[15].Axis[5].Pos3.Reached := FALSE;
   AxisStore[15].Axis[5].Pos4.Position := 0.0;
   AxisStore[15].Axis[5].Pos4.Speed := 0;
   AxisStore[15].Axis[5].Pos4.Reached := FALSE;
   AxisStore[15].Axis[5].Pos5.Position := 0.0;
   AxisStore[15].Axis[5].Pos5.Speed := 0;
   AxisStore[15].Axis[5].Pos5.Reached := FALSE;
   AxisStore[15].Axis[5].Pos6.Position := 0.0;
   AxisStore[15].Axis[5].Pos6.Speed := 0;
   AxisStore[15].Axis[5].Pos6.Reached := FALSE;
   AxisStore[15].Axis[5].Pos7.Position := 0.0;
   AxisStore[15].Axis[5].Pos7.Speed := 0;
   AxisStore[15].Axis[5].Pos7.Reached := FALSE;
   AxisStore[15].Axis[5].Pos8.Position := 0.0;
   AxisStore[15].Axis[5].Pos8.Speed := 0;
   AxisStore[15].Axis[5].Pos8.Reached := FALSE;
   AxisStore[15].Axis[5].Pos9.Position := 0.0;
   AxisStore[15].Axis[5].Pos9.Speed := 0;
   AxisStore[15].Axis[5].Pos9.Reached := FALSE;
   AxisStore[15].Axis[5].Pos10.Position := 0.0;
   AxisStore[15].Axis[5].Pos10.Speed := 0;
   AxisStore[15].Axis[5].Pos10.Reached := FALSE;
   AxisStore[15].Axis[5].Pos11.Position := 0.0;
   AxisStore[15].Axis[5].Pos11.Speed := 0;
   AxisStore[15].Axis[5].Pos11.Reached := FALSE;
   AxisStore[15].Axis[5].Pos12.Position := 0.0;
   AxisStore[15].Axis[5].Pos12.Speed := 0;
   AxisStore[15].Axis[5].Pos12.Reached := FALSE;
   AxisStore[15].Axis[5].Pos13.Position := 0.0;
   AxisStore[15].Axis[5].Pos13.Speed := 0;
   AxisStore[15].Axis[5].Pos13.Reached := FALSE;
   AxisStore[15].Axis[5].Pos14.Position := 0.0;
   AxisStore[15].Axis[5].Pos14.Speed := 0;
   AxisStore[15].Axis[5].Pos14.Reached := FALSE;
   AxisStore[15].Axis[5].Pos15.Position := 0.0;
   AxisStore[15].Axis[5].Pos15.Speed := 0;
   AxisStore[15].Axis[5].Pos15.Reached := FALSE;
   AxisStore[15].Axis[5].Pos16.Position := 0.0;
   AxisStore[15].Axis[5].Pos16.Speed := 0;
   AxisStore[15].Axis[5].Pos16.Reached := FALSE;
   AxisStore[15].Axis[5].Pos17.Position := 0.0;
   AxisStore[15].Axis[5].Pos17.Speed := 0;
   AxisStore[15].Axis[5].Pos17.Reached := FALSE;
   AxisStore[15].Axis[5].Pos18.Position := 0.0;
   AxisStore[15].Axis[5].Pos18.Speed := 0;
   AxisStore[15].Axis[5].Pos18.Reached := FALSE;
   AxisStore[15].Axis[5].Pos19.Position := 0.0;
   AxisStore[15].Axis[5].Pos19.Speed := 0;
   AxisStore[15].Axis[5].Pos19.Reached := FALSE;
   AxisStore[15].Axis[5].Pos20.Position := 0.0;
   AxisStore[15].Axis[5].Pos20.Speed := 0;
   AxisStore[15].Axis[5].Pos20.Reached := FALSE;
   AxisStore[15].Axis[5].Pos21.Position := 0.0;
   AxisStore[15].Axis[5].Pos21.Speed := 0;
   AxisStore[15].Axis[5].Pos21.Reached := FALSE;
   AxisStore[15].Axis[5].Pos22.Position := 0.0;
   AxisStore[15].Axis[5].Pos22.Speed := 0;
   AxisStore[15].Axis[5].Pos22.Reached := FALSE;
   AxisStore[15].Axis[5].Pos23.Position := 0.0;
   AxisStore[15].Axis[5].Pos23.Speed := 0;
   AxisStore[15].Axis[5].Pos23.Reached := FALSE;
   AxisStore[15].Axis[5].Pos24.Position := 0.0;
   AxisStore[15].Axis[5].Pos24.Speed := 0;
   AxisStore[15].Axis[5].Pos24.Reached := FALSE;
   AxisStore[15].Axis[5].Pos25.Position := 0.0;
   AxisStore[15].Axis[5].Pos25.Speed := 0;
   AxisStore[15].Axis[5].Pos25.Reached := FALSE;
   AxisStore[15].Axis[5].Pos26.Position := 0.0;
   AxisStore[15].Axis[5].Pos26.Speed := 0;
   AxisStore[15].Axis[5].Pos26.Reached := FALSE;
   AxisStore[15].Axis[5].Pos27.Position := 0.0;
   AxisStore[15].Axis[5].Pos27.Speed := 0;
   AxisStore[15].Axis[5].Pos27.Reached := FALSE;
   AxisStore[15].Axis[5].Pos28.Position := 0.0;
   AxisStore[15].Axis[5].Pos28.Speed := 0;
   AxisStore[15].Axis[5].Pos28.Reached := FALSE;
   AxisStore[15].Axis[5].Pos29.Position := 0.0;
   AxisStore[15].Axis[5].Pos29.Speed := 0;
   AxisStore[15].Axis[5].Pos29.Reached := FALSE;
   AxisStore[15].Axis[5].Pos30.Position := 0.0;
   AxisStore[15].Axis[5].Pos30.Speed := 0;
   AxisStore[15].Axis[5].Pos30.Reached := FALSE;
   AxisStore[15].Axis[6].Pos1.Position := 0.0;
   AxisStore[15].Axis[6].Pos1.Speed := 0;
   AxisStore[15].Axis[6].Pos1.Reached := FALSE;
   AxisStore[15].Axis[6].Pos2.Position := 0.0;
   AxisStore[15].Axis[6].Pos2.Speed := 0;
   AxisStore[15].Axis[6].Pos2.Reached := FALSE;
   AxisStore[15].Axis[6].Pos3.Position := 0.0;
   AxisStore[15].Axis[6].Pos3.Speed := 0;
   AxisStore[15].Axis[6].Pos3.Reached := FALSE;
   AxisStore[15].Axis[6].Pos4.Position := 0.0;
   AxisStore[15].Axis[6].Pos4.Speed := 0;
   AxisStore[15].Axis[6].Pos4.Reached := FALSE;
   AxisStore[15].Axis[6].Pos5.Position := 0.0;
   AxisStore[15].Axis[6].Pos5.Speed := 0;
   AxisStore[15].Axis[6].Pos5.Reached := FALSE;
   AxisStore[15].Axis[6].Pos6.Position := 0.0;
   AxisStore[15].Axis[6].Pos6.Speed := 0;
   AxisStore[15].Axis[6].Pos6.Reached := FALSE;
   AxisStore[15].Axis[6].Pos7.Position := 0.0;
   AxisStore[15].Axis[6].Pos7.Speed := 0;
   AxisStore[15].Axis[6].Pos7.Reached := FALSE;
   AxisStore[15].Axis[6].Pos8.Position := 0.0;
   AxisStore[15].Axis[6].Pos8.Speed := 0;
   AxisStore[15].Axis[6].Pos8.Reached := FALSE;
   AxisStore[15].Axis[6].Pos9.Position := 0.0;
   AxisStore[15].Axis[6].Pos9.Speed := 0;
   AxisStore[15].Axis[6].Pos9.Reached := FALSE;
   AxisStore[15].Axis[6].Pos10.Position := 0.0;
   AxisStore[15].Axis[6].Pos10.Speed := 0;
   AxisStore[15].Axis[6].Pos10.Reached := FALSE;
   AxisStore[15].Axis[6].Pos11.Position := 0.0;
   AxisStore[15].Axis[6].Pos11.Speed := 0;
   AxisStore[15].Axis[6].Pos11.Reached := FALSE;
   AxisStore[15].Axis[6].Pos12.Position := 0.0;
   AxisStore[15].Axis[6].Pos12.Speed := 0;
   AxisStore[15].Axis[6].Pos12.Reached := FALSE;
   AxisStore[15].Axis[6].Pos13.Position := 0.0;
   AxisStore[15].Axis[6].Pos13.Speed := 0;
   AxisStore[15].Axis[6].Pos13.Reached := FALSE;
   AxisStore[15].Axis[6].Pos14.Position := 0.0;
   AxisStore[15].Axis[6].Pos14.Speed := 0;
   AxisStore[15].Axis[6].Pos14.Reached := FALSE;
   AxisStore[15].Axis[6].Pos15.Position := 0.0;
   AxisStore[15].Axis[6].Pos15.Speed := 0;
   AxisStore[15].Axis[6].Pos15.Reached := FALSE;
   AxisStore[15].Axis[6].Pos16.Position := 0.0;
   AxisStore[15].Axis[6].Pos16.Speed := 0;
   AxisStore[15].Axis[6].Pos16.Reached := FALSE;
   AxisStore[15].Axis[6].Pos17.Position := 0.0;
   AxisStore[15].Axis[6].Pos17.Speed := 0;
   AxisStore[15].Axis[6].Pos17.Reached := FALSE;
   AxisStore[15].Axis[6].Pos18.Position := 0.0;
   AxisStore[15].Axis[6].Pos18.Speed := 0;
   AxisStore[15].Axis[6].Pos18.Reached := FALSE;
   AxisStore[15].Axis[6].Pos19.Position := 0.0;
   AxisStore[15].Axis[6].Pos19.Speed := 0;
   AxisStore[15].Axis[6].Pos19.Reached := FALSE;
   AxisStore[15].Axis[6].Pos20.Position := 0.0;
   AxisStore[15].Axis[6].Pos20.Speed := 0;
   AxisStore[15].Axis[6].Pos20.Reached := FALSE;
   AxisStore[15].Axis[6].Pos21.Position := 0.0;
   AxisStore[15].Axis[6].Pos21.Speed := 0;
   AxisStore[15].Axis[6].Pos21.Reached := FALSE;
   AxisStore[15].Axis[6].Pos22.Position := 0.0;
   AxisStore[15].Axis[6].Pos22.Speed := 0;
   AxisStore[15].Axis[6].Pos22.Reached := FALSE;
   AxisStore[15].Axis[6].Pos23.Position := 0.0;
   AxisStore[15].Axis[6].Pos23.Speed := 0;
   AxisStore[15].Axis[6].Pos23.Reached := FALSE;
   AxisStore[15].Axis[6].Pos24.Position := 0.0;
   AxisStore[15].Axis[6].Pos24.Speed := 0;
   AxisStore[15].Axis[6].Pos24.Reached := FALSE;
   AxisStore[15].Axis[6].Pos25.Position := 0.0;
   AxisStore[15].Axis[6].Pos25.Speed := 0;
   AxisStore[15].Axis[6].Pos25.Reached := FALSE;
   AxisStore[15].Axis[6].Pos26.Position := 0.0;
   AxisStore[15].Axis[6].Pos26.Speed := 0;
   AxisStore[15].Axis[6].Pos26.Reached := FALSE;
   AxisStore[15].Axis[6].Pos27.Position := 0.0;
   AxisStore[15].Axis[6].Pos27.Speed := 0;
   AxisStore[15].Axis[6].Pos27.Reached := FALSE;
   AxisStore[15].Axis[6].Pos28.Position := 0.0;
   AxisStore[15].Axis[6].Pos28.Speed := 0;
   AxisStore[15].Axis[6].Pos28.Reached := FALSE;
   AxisStore[15].Axis[6].Pos29.Position := 0.0;
   AxisStore[15].Axis[6].Pos29.Speed := 0;
   AxisStore[15].Axis[6].Pos29.Reached := FALSE;
   AxisStore[15].Axis[6].Pos30.Position := 0.0;
   AxisStore[15].Axis[6].Pos30.Speed := 0;
   AxisStore[15].Axis[6].Pos30.Reached := FALSE;
   AxisStore[15].Axis[7].Pos1.Position := 0.0;
   AxisStore[15].Axis[7].Pos1.Speed := 0;
   AxisStore[15].Axis[7].Pos1.Reached := FALSE;
   AxisStore[15].Axis[7].Pos2.Position := 0.0;
   AxisStore[15].Axis[7].Pos2.Speed := 0;
   AxisStore[15].Axis[7].Pos2.Reached := FALSE;
   AxisStore[15].Axis[7].Pos3.Position := 0.0;
   AxisStore[15].Axis[7].Pos3.Speed := 0;
   AxisStore[15].Axis[7].Pos3.Reached := FALSE;
   AxisStore[15].Axis[7].Pos4.Position := 0.0;
   AxisStore[15].Axis[7].Pos4.Speed := 0;
   AxisStore[15].Axis[7].Pos4.Reached := FALSE;
   AxisStore[15].Axis[7].Pos5.Position := 0.0;
   AxisStore[15].Axis[7].Pos5.Speed := 0;
   AxisStore[15].Axis[7].Pos5.Reached := FALSE;
   AxisStore[15].Axis[7].Pos6.Position := 0.0;
   AxisStore[15].Axis[7].Pos6.Speed := 0;
   AxisStore[15].Axis[7].Pos6.Reached := FALSE;
   AxisStore[15].Axis[7].Pos7.Position := 0.0;
   AxisStore[15].Axis[7].Pos7.Speed := 0;
   AxisStore[15].Axis[7].Pos7.Reached := FALSE;
   AxisStore[15].Axis[7].Pos8.Position := 0.0;
   AxisStore[15].Axis[7].Pos8.Speed := 0;
   AxisStore[15].Axis[7].Pos8.Reached := FALSE;
   AxisStore[15].Axis[7].Pos9.Position := 0.0;
   AxisStore[15].Axis[7].Pos9.Speed := 0;
   AxisStore[15].Axis[7].Pos9.Reached := FALSE;
   AxisStore[15].Axis[7].Pos10.Position := 0.0;
   AxisStore[15].Axis[7].Pos10.Speed := 0;
   AxisStore[15].Axis[7].Pos10.Reached := FALSE;
   AxisStore[15].Axis[7].Pos11.Position := 0.0;
   AxisStore[15].Axis[7].Pos11.Speed := 0;
   AxisStore[15].Axis[7].Pos11.Reached := FALSE;
   AxisStore[15].Axis[7].Pos12.Position := 0.0;
   AxisStore[15].Axis[7].Pos12.Speed := 0;
   AxisStore[15].Axis[7].Pos12.Reached := FALSE;
   AxisStore[15].Axis[7].Pos13.Position := 0.0;
   AxisStore[15].Axis[7].Pos13.Speed := 0;
   AxisStore[15].Axis[7].Pos13.Reached := FALSE;
   AxisStore[15].Axis[7].Pos14.Position := 0.0;
   AxisStore[15].Axis[7].Pos14.Speed := 0;
   AxisStore[15].Axis[7].Pos14.Reached := FALSE;
   AxisStore[15].Axis[7].Pos15.Position := 0.0;
   AxisStore[15].Axis[7].Pos15.Speed := 0;
   AxisStore[15].Axis[7].Pos15.Reached := FALSE;
   AxisStore[15].Axis[7].Pos16.Position := 0.0;
   AxisStore[15].Axis[7].Pos16.Speed := 0;
   AxisStore[15].Axis[7].Pos16.Reached := FALSE;
   AxisStore[15].Axis[7].Pos17.Position := 0.0;
   AxisStore[15].Axis[7].Pos17.Speed := 0;
   AxisStore[15].Axis[7].Pos17.Reached := FALSE;
   AxisStore[15].Axis[7].Pos18.Position := 0.0;
   AxisStore[15].Axis[7].Pos18.Speed := 0;
   AxisStore[15].Axis[7].Pos18.Reached := FALSE;
   AxisStore[15].Axis[7].Pos19.Position := 0.0;
   AxisStore[15].Axis[7].Pos19.Speed := 0;
   AxisStore[15].Axis[7].Pos19.Reached := FALSE;
   AxisStore[15].Axis[7].Pos20.Position := 0.0;
   AxisStore[15].Axis[7].Pos20.Speed := 0;
   AxisStore[15].Axis[7].Pos20.Reached := FALSE;
   AxisStore[15].Axis[7].Pos21.Position := 0.0;
   AxisStore[15].Axis[7].Pos21.Speed := 0;
   AxisStore[15].Axis[7].Pos21.Reached := FALSE;
   AxisStore[15].Axis[7].Pos22.Position := 0.0;
   AxisStore[15].Axis[7].Pos22.Speed := 0;
   AxisStore[15].Axis[7].Pos22.Reached := FALSE;
   AxisStore[15].Axis[7].Pos23.Position := 0.0;
   AxisStore[15].Axis[7].Pos23.Speed := 0;
   AxisStore[15].Axis[7].Pos23.Reached := FALSE;
   AxisStore[15].Axis[7].Pos24.Position := 0.0;
   AxisStore[15].Axis[7].Pos24.Speed := 0;
   AxisStore[15].Axis[7].Pos24.Reached := FALSE;
   AxisStore[15].Axis[7].Pos25.Position := 0.0;
   AxisStore[15].Axis[7].Pos25.Speed := 0;
   AxisStore[15].Axis[7].Pos25.Reached := FALSE;
   AxisStore[15].Axis[7].Pos26.Position := 0.0;
   AxisStore[15].Axis[7].Pos26.Speed := 0;
   AxisStore[15].Axis[7].Pos26.Reached := FALSE;
   AxisStore[15].Axis[7].Pos27.Position := 0.0;
   AxisStore[15].Axis[7].Pos27.Speed := 0;
   AxisStore[15].Axis[7].Pos27.Reached := FALSE;
   AxisStore[15].Axis[7].Pos28.Position := 0.0;
   AxisStore[15].Axis[7].Pos28.Speed := 0;
   AxisStore[15].Axis[7].Pos28.Reached := FALSE;
   AxisStore[15].Axis[7].Pos29.Position := 0.0;
   AxisStore[15].Axis[7].Pos29.Speed := 0;
   AxisStore[15].Axis[7].Pos29.Reached := FALSE;
   AxisStore[15].Axis[7].Pos30.Position := 0.0;
   AxisStore[15].Axis[7].Pos30.Speed := 0;
   AxisStore[15].Axis[7].Pos30.Reached := FALSE;
   AxisStore[15].Axis[8].Pos1.Position := 0.0;
   AxisStore[15].Axis[8].Pos1.Speed := 0;
   AxisStore[15].Axis[8].Pos1.Reached := FALSE;
   AxisStore[15].Axis[8].Pos2.Position := 0.0;
   AxisStore[15].Axis[8].Pos2.Speed := 0;
   AxisStore[15].Axis[8].Pos2.Reached := FALSE;
   AxisStore[15].Axis[8].Pos3.Position := 0.0;
   AxisStore[15].Axis[8].Pos3.Speed := 0;
   AxisStore[15].Axis[8].Pos3.Reached := FALSE;
   AxisStore[15].Axis[8].Pos4.Position := 0.0;
   AxisStore[15].Axis[8].Pos4.Speed := 0;
   AxisStore[15].Axis[8].Pos4.Reached := FALSE;
   AxisStore[15].Axis[8].Pos5.Position := 0.0;
   AxisStore[15].Axis[8].Pos5.Speed := 0;
   AxisStore[15].Axis[8].Pos5.Reached := FALSE;
   AxisStore[15].Axis[8].Pos6.Position := 0.0;
   AxisStore[15].Axis[8].Pos6.Speed := 0;
   AxisStore[15].Axis[8].Pos6.Reached := FALSE;
   AxisStore[15].Axis[8].Pos7.Position := 0.0;
   AxisStore[15].Axis[8].Pos7.Speed := 0;
   AxisStore[15].Axis[8].Pos7.Reached := FALSE;
   AxisStore[15].Axis[8].Pos8.Position := 0.0;
   AxisStore[15].Axis[8].Pos8.Speed := 0;
   AxisStore[15].Axis[8].Pos8.Reached := FALSE;
   AxisStore[15].Axis[8].Pos9.Position := 0.0;
   AxisStore[15].Axis[8].Pos9.Speed := 0;
   AxisStore[15].Axis[8].Pos9.Reached := FALSE;
   AxisStore[15].Axis[8].Pos10.Position := 0.0;
   AxisStore[15].Axis[8].Pos10.Speed := 0;
   AxisStore[15].Axis[8].Pos10.Reached := FALSE;
   AxisStore[15].Axis[8].Pos11.Position := 0.0;
   AxisStore[15].Axis[8].Pos11.Speed := 0;
   AxisStore[15].Axis[8].Pos11.Reached := FALSE;
   AxisStore[15].Axis[8].Pos12.Position := 0.0;
   AxisStore[15].Axis[8].Pos12.Speed := 0;
   AxisStore[15].Axis[8].Pos12.Reached := FALSE;
   AxisStore[15].Axis[8].Pos13.Position := 0.0;
   AxisStore[15].Axis[8].Pos13.Speed := 0;
   AxisStore[15].Axis[8].Pos13.Reached := FALSE;
   AxisStore[15].Axis[8].Pos14.Position := 0.0;
   AxisStore[15].Axis[8].Pos14.Speed := 0;
   AxisStore[15].Axis[8].Pos14.Reached := FALSE;
   AxisStore[15].Axis[8].Pos15.Position := 0.0;
   AxisStore[15].Axis[8].Pos15.Speed := 0;
   AxisStore[15].Axis[8].Pos15.Reached := FALSE;
   AxisStore[15].Axis[8].Pos16.Position := 0.0;
   AxisStore[15].Axis[8].Pos16.Speed := 0;
   AxisStore[15].Axis[8].Pos16.Reached := FALSE;
   AxisStore[15].Axis[8].Pos17.Position := 0.0;
   AxisStore[15].Axis[8].Pos17.Speed := 0;
   AxisStore[15].Axis[8].Pos17.Reached := FALSE;
   AxisStore[15].Axis[8].Pos18.Position := 0.0;
   AxisStore[15].Axis[8].Pos18.Speed := 0;
   AxisStore[15].Axis[8].Pos18.Reached := FALSE;
   AxisStore[15].Axis[8].Pos19.Position := 0.0;
   AxisStore[15].Axis[8].Pos19.Speed := 0;
   AxisStore[15].Axis[8].Pos19.Reached := FALSE;
   AxisStore[15].Axis[8].Pos20.Position := 0.0;
   AxisStore[15].Axis[8].Pos20.Speed := 0;
   AxisStore[15].Axis[8].Pos20.Reached := FALSE;
   AxisStore[15].Axis[8].Pos21.Position := 0.0;
   AxisStore[15].Axis[8].Pos21.Speed := 0;
   AxisStore[15].Axis[8].Pos21.Reached := FALSE;
   AxisStore[15].Axis[8].Pos22.Position := 0.0;
   AxisStore[15].Axis[8].Pos22.Speed := 0;
   AxisStore[15].Axis[8].Pos22.Reached := FALSE;
   AxisStore[15].Axis[8].Pos23.Position := 0.0;
   AxisStore[15].Axis[8].Pos23.Speed := 0;
   AxisStore[15].Axis[8].Pos23.Reached := FALSE;
   AxisStore[15].Axis[8].Pos24.Position := 0.0;
   AxisStore[15].Axis[8].Pos24.Speed := 0;
   AxisStore[15].Axis[8].Pos24.Reached := FALSE;
   AxisStore[15].Axis[8].Pos25.Position := 0.0;
   AxisStore[15].Axis[8].Pos25.Speed := 0;
   AxisStore[15].Axis[8].Pos25.Reached := FALSE;
   AxisStore[15].Axis[8].Pos26.Position := 0.0;
   AxisStore[15].Axis[8].Pos26.Speed := 0;
   AxisStore[15].Axis[8].Pos26.Reached := FALSE;
   AxisStore[15].Axis[8].Pos27.Position := 0.0;
   AxisStore[15].Axis[8].Pos27.Speed := 0;
   AxisStore[15].Axis[8].Pos27.Reached := FALSE;
   AxisStore[15].Axis[8].Pos28.Position := 0.0;
   AxisStore[15].Axis[8].Pos28.Speed := 0;
   AxisStore[15].Axis[8].Pos28.Reached := FALSE;
   AxisStore[15].Axis[8].Pos29.Position := 0.0;
   AxisStore[15].Axis[8].Pos29.Speed := 0;
   AxisStore[15].Axis[8].Pos29.Reached := FALSE;
   AxisStore[15].Axis[8].Pos30.Position := 0.0;
   AxisStore[15].Axis[8].Pos30.Speed := 0;
   AxisStore[15].Axis[8].Pos30.Reached := FALSE;
   AxisStore[15].Axis[9].Pos1.Position := 0.0;
   AxisStore[15].Axis[9].Pos1.Speed := 0;
   AxisStore[15].Axis[9].Pos1.Reached := FALSE;
   AxisStore[15].Axis[9].Pos2.Position := 0.0;
   AxisStore[15].Axis[9].Pos2.Speed := 0;
   AxisStore[15].Axis[9].Pos2.Reached := FALSE;
   AxisStore[15].Axis[9].Pos3.Position := 0.0;
   AxisStore[15].Axis[9].Pos3.Speed := 0;
   AxisStore[15].Axis[9].Pos3.Reached := FALSE;
   AxisStore[15].Axis[9].Pos4.Position := 0.0;
   AxisStore[15].Axis[9].Pos4.Speed := 0;
   AxisStore[15].Axis[9].Pos4.Reached := FALSE;
   AxisStore[15].Axis[9].Pos5.Position := 0.0;
   AxisStore[15].Axis[9].Pos5.Speed := 0;
   AxisStore[15].Axis[9].Pos5.Reached := FALSE;
   AxisStore[15].Axis[9].Pos6.Position := 0.0;
   AxisStore[15].Axis[9].Pos6.Speed := 0;
   AxisStore[15].Axis[9].Pos6.Reached := FALSE;
   AxisStore[15].Axis[9].Pos7.Position := 0.0;
   AxisStore[15].Axis[9].Pos7.Speed := 0;
   AxisStore[15].Axis[9].Pos7.Reached := FALSE;
   AxisStore[15].Axis[9].Pos8.Position := 0.0;
   AxisStore[15].Axis[9].Pos8.Speed := 0;
   AxisStore[15].Axis[9].Pos8.Reached := FALSE;
   AxisStore[15].Axis[9].Pos9.Position := 0.0;
   AxisStore[15].Axis[9].Pos9.Speed := 0;
   AxisStore[15].Axis[9].Pos9.Reached := FALSE;
   AxisStore[15].Axis[9].Pos10.Position := 0.0;
   AxisStore[15].Axis[9].Pos10.Speed := 0;
   AxisStore[15].Axis[9].Pos10.Reached := FALSE;
   AxisStore[15].Axis[9].Pos11.Position := 0.0;
   AxisStore[15].Axis[9].Pos11.Speed := 0;
   AxisStore[15].Axis[9].Pos11.Reached := FALSE;
   AxisStore[15].Axis[9].Pos12.Position := 0.0;
   AxisStore[15].Axis[9].Pos12.Speed := 0;
   AxisStore[15].Axis[9].Pos12.Reached := FALSE;
   AxisStore[15].Axis[9].Pos13.Position := 0.0;
   AxisStore[15].Axis[9].Pos13.Speed := 0;
   AxisStore[15].Axis[9].Pos13.Reached := FALSE;
   AxisStore[15].Axis[9].Pos14.Position := 0.0;
   AxisStore[15].Axis[9].Pos14.Speed := 0;
   AxisStore[15].Axis[9].Pos14.Reached := FALSE;
   AxisStore[15].Axis[9].Pos15.Position := 0.0;
   AxisStore[15].Axis[9].Pos15.Speed := 0;
   AxisStore[15].Axis[9].Pos15.Reached := FALSE;
   AxisStore[15].Axis[9].Pos16.Position := 0.0;
   AxisStore[15].Axis[9].Pos16.Speed := 0;
   AxisStore[15].Axis[9].Pos16.Reached := FALSE;
   AxisStore[15].Axis[9].Pos17.Position := 0.0;
   AxisStore[15].Axis[9].Pos17.Speed := 0;
   AxisStore[15].Axis[9].Pos17.Reached := FALSE;
   AxisStore[15].Axis[9].Pos18.Position := 0.0;
   AxisStore[15].Axis[9].Pos18.Speed := 0;
   AxisStore[15].Axis[9].Pos18.Reached := FALSE;
   AxisStore[15].Axis[9].Pos19.Position := 0.0;
   AxisStore[15].Axis[9].Pos19.Speed := 0;
   AxisStore[15].Axis[9].Pos19.Reached := FALSE;
   AxisStore[15].Axis[9].Pos20.Position := 0.0;
   AxisStore[15].Axis[9].Pos20.Speed := 0;
   AxisStore[15].Axis[9].Pos20.Reached := FALSE;
   AxisStore[15].Axis[9].Pos21.Position := 0.0;
   AxisStore[15].Axis[9].Pos21.Speed := 0;
   AxisStore[15].Axis[9].Pos21.Reached := FALSE;
   AxisStore[15].Axis[9].Pos22.Position := 0.0;
   AxisStore[15].Axis[9].Pos22.Speed := 0;
   AxisStore[15].Axis[9].Pos22.Reached := FALSE;
   AxisStore[15].Axis[9].Pos23.Position := 0.0;
   AxisStore[15].Axis[9].Pos23.Speed := 0;
   AxisStore[15].Axis[9].Pos23.Reached := FALSE;
   AxisStore[15].Axis[9].Pos24.Position := 0.0;
   AxisStore[15].Axis[9].Pos24.Speed := 0;
   AxisStore[15].Axis[9].Pos24.Reached := FALSE;
   AxisStore[15].Axis[9].Pos25.Position := 0.0;
   AxisStore[15].Axis[9].Pos25.Speed := 0;
   AxisStore[15].Axis[9].Pos25.Reached := FALSE;
   AxisStore[15].Axis[9].Pos26.Position := 0.0;
   AxisStore[15].Axis[9].Pos26.Speed := 0;
   AxisStore[15].Axis[9].Pos26.Reached := FALSE;
   AxisStore[15].Axis[9].Pos27.Position := 0.0;
   AxisStore[15].Axis[9].Pos27.Speed := 0;
   AxisStore[15].Axis[9].Pos27.Reached := FALSE;
   AxisStore[15].Axis[9].Pos28.Position := 0.0;
   AxisStore[15].Axis[9].Pos28.Speed := 0;
   AxisStore[15].Axis[9].Pos28.Reached := FALSE;
   AxisStore[15].Axis[9].Pos29.Position := 0.0;
   AxisStore[15].Axis[9].Pos29.Speed := 0;
   AxisStore[15].Axis[9].Pos29.Reached := FALSE;
   AxisStore[15].Axis[9].Pos30.Position := 0.0;
   AxisStore[15].Axis[9].Pos30.Speed := 0;
   AxisStore[15].Axis[9].Pos30.Reached := FALSE;
   AxisStore[15].Axis[10].Pos1.Position := 0.0;
   AxisStore[15].Axis[10].Pos1.Speed := 0;
   AxisStore[15].Axis[10].Pos1.Reached := FALSE;
   AxisStore[15].Axis[10].Pos2.Position := 0.0;
   AxisStore[15].Axis[10].Pos2.Speed := 0;
   AxisStore[15].Axis[10].Pos2.Reached := FALSE;
   AxisStore[15].Axis[10].Pos3.Position := 0.0;
   AxisStore[15].Axis[10].Pos3.Speed := 0;
   AxisStore[15].Axis[10].Pos3.Reached := FALSE;
   AxisStore[15].Axis[10].Pos4.Position := 0.0;
   AxisStore[15].Axis[10].Pos4.Speed := 0;
   AxisStore[15].Axis[10].Pos4.Reached := FALSE;
   AxisStore[15].Axis[10].Pos5.Position := 0.0;
   AxisStore[15].Axis[10].Pos5.Speed := 0;
   AxisStore[15].Axis[10].Pos5.Reached := FALSE;
   AxisStore[15].Axis[10].Pos6.Position := 0.0;
   AxisStore[15].Axis[10].Pos6.Speed := 0;
   AxisStore[15].Axis[10].Pos6.Reached := FALSE;
   AxisStore[15].Axis[10].Pos7.Position := 0.0;
   AxisStore[15].Axis[10].Pos7.Speed := 0;
   AxisStore[15].Axis[10].Pos7.Reached := FALSE;
   AxisStore[15].Axis[10].Pos8.Position := 0.0;
   AxisStore[15].Axis[10].Pos8.Speed := 0;
   AxisStore[15].Axis[10].Pos8.Reached := FALSE;
   AxisStore[15].Axis[10].Pos9.Position := 0.0;
   AxisStore[15].Axis[10].Pos9.Speed := 0;
   AxisStore[15].Axis[10].Pos9.Reached := FALSE;
   AxisStore[15].Axis[10].Pos10.Position := 0.0;
   AxisStore[15].Axis[10].Pos10.Speed := 0;
   AxisStore[15].Axis[10].Pos10.Reached := FALSE;
   AxisStore[15].Axis[10].Pos11.Position := 0.0;
   AxisStore[15].Axis[10].Pos11.Speed := 0;
   AxisStore[15].Axis[10].Pos11.Reached := FALSE;
   AxisStore[15].Axis[10].Pos12.Position := 0.0;
   AxisStore[15].Axis[10].Pos12.Speed := 0;
   AxisStore[15].Axis[10].Pos12.Reached := FALSE;
   AxisStore[15].Axis[10].Pos13.Position := 0.0;
   AxisStore[15].Axis[10].Pos13.Speed := 0;
   AxisStore[15].Axis[10].Pos13.Reached := FALSE;
   AxisStore[15].Axis[10].Pos14.Position := 0.0;
   AxisStore[15].Axis[10].Pos14.Speed := 0;
   AxisStore[15].Axis[10].Pos14.Reached := FALSE;
   AxisStore[15].Axis[10].Pos15.Position := 0.0;
   AxisStore[15].Axis[10].Pos15.Speed := 0;
   AxisStore[15].Axis[10].Pos15.Reached := FALSE;
   AxisStore[15].Axis[10].Pos16.Position := 0.0;
   AxisStore[15].Axis[10].Pos16.Speed := 0;
   AxisStore[15].Axis[10].Pos16.Reached := FALSE;
   AxisStore[15].Axis[10].Pos17.Position := 0.0;
   AxisStore[15].Axis[10].Pos17.Speed := 0;
   AxisStore[15].Axis[10].Pos17.Reached := FALSE;
   AxisStore[15].Axis[10].Pos18.Position := 0.0;
   AxisStore[15].Axis[10].Pos18.Speed := 0;
   AxisStore[15].Axis[10].Pos18.Reached := FALSE;
   AxisStore[15].Axis[10].Pos19.Position := 0.0;
   AxisStore[15].Axis[10].Pos19.Speed := 0;
   AxisStore[15].Axis[10].Pos19.Reached := FALSE;
   AxisStore[15].Axis[10].Pos20.Position := 0.0;
   AxisStore[15].Axis[10].Pos20.Speed := 0;
   AxisStore[15].Axis[10].Pos20.Reached := FALSE;
   AxisStore[15].Axis[10].Pos21.Position := 0.0;
   AxisStore[15].Axis[10].Pos21.Speed := 0;
   AxisStore[15].Axis[10].Pos21.Reached := FALSE;
   AxisStore[15].Axis[10].Pos22.Position := 0.0;
   AxisStore[15].Axis[10].Pos22.Speed := 0;
   AxisStore[15].Axis[10].Pos22.Reached := FALSE;
   AxisStore[15].Axis[10].Pos23.Position := 0.0;
   AxisStore[15].Axis[10].Pos23.Speed := 0;
   AxisStore[15].Axis[10].Pos23.Reached := FALSE;
   AxisStore[15].Axis[10].Pos24.Position := 0.0;
   AxisStore[15].Axis[10].Pos24.Speed := 0;
   AxisStore[15].Axis[10].Pos24.Reached := FALSE;
   AxisStore[15].Axis[10].Pos25.Position := 0.0;
   AxisStore[15].Axis[10].Pos25.Speed := 0;
   AxisStore[15].Axis[10].Pos25.Reached := FALSE;
   AxisStore[15].Axis[10].Pos26.Position := 0.0;
   AxisStore[15].Axis[10].Pos26.Speed := 0;
   AxisStore[15].Axis[10].Pos26.Reached := FALSE;
   AxisStore[15].Axis[10].Pos27.Position := 0.0;
   AxisStore[15].Axis[10].Pos27.Speed := 0;
   AxisStore[15].Axis[10].Pos27.Reached := FALSE;
   AxisStore[15].Axis[10].Pos28.Position := 0.0;
   AxisStore[15].Axis[10].Pos28.Speed := 0;
   AxisStore[15].Axis[10].Pos28.Reached := FALSE;
   AxisStore[15].Axis[10].Pos29.Position := 0.0;
   AxisStore[15].Axis[10].Pos29.Speed := 0;
   AxisStore[15].Axis[10].Pos29.Reached := FALSE;
   AxisStore[15].Axis[10].Pos30.Position := 0.0;
   AxisStore[15].Axis[10].Pos30.Speed := 0;
   AxisStore[15].Axis[10].Pos30.Reached := FALSE;
   AxisStore[15].Axis[11].Pos1.Position := 0.0;
   AxisStore[15].Axis[11].Pos1.Speed := 0;
   AxisStore[15].Axis[11].Pos1.Reached := FALSE;
   AxisStore[15].Axis[11].Pos2.Position := 0.0;
   AxisStore[15].Axis[11].Pos2.Speed := 0;
   AxisStore[15].Axis[11].Pos2.Reached := FALSE;
   AxisStore[15].Axis[11].Pos3.Position := 0.0;
   AxisStore[15].Axis[11].Pos3.Speed := 0;
   AxisStore[15].Axis[11].Pos3.Reached := FALSE;
   AxisStore[15].Axis[11].Pos4.Position := 0.0;
   AxisStore[15].Axis[11].Pos4.Speed := 0;
   AxisStore[15].Axis[11].Pos4.Reached := FALSE;
   AxisStore[15].Axis[11].Pos5.Position := 0.0;
   AxisStore[15].Axis[11].Pos5.Speed := 0;
   AxisStore[15].Axis[11].Pos5.Reached := FALSE;
   AxisStore[15].Axis[11].Pos6.Position := 0.0;
   AxisStore[15].Axis[11].Pos6.Speed := 0;
   AxisStore[15].Axis[11].Pos6.Reached := FALSE;
   AxisStore[15].Axis[11].Pos7.Position := 0.0;
   AxisStore[15].Axis[11].Pos7.Speed := 0;
   AxisStore[15].Axis[11].Pos7.Reached := FALSE;
   AxisStore[15].Axis[11].Pos8.Position := 0.0;
   AxisStore[15].Axis[11].Pos8.Speed := 0;
   AxisStore[15].Axis[11].Pos8.Reached := FALSE;
   AxisStore[15].Axis[11].Pos9.Position := 0.0;
   AxisStore[15].Axis[11].Pos9.Speed := 0;
   AxisStore[15].Axis[11].Pos9.Reached := FALSE;
   AxisStore[15].Axis[11].Pos10.Position := 0.0;
   AxisStore[15].Axis[11].Pos10.Speed := 0;
   AxisStore[15].Axis[11].Pos10.Reached := FALSE;
   AxisStore[15].Axis[11].Pos11.Position := 0.0;
   AxisStore[15].Axis[11].Pos11.Speed := 0;
   AxisStore[15].Axis[11].Pos11.Reached := FALSE;
   AxisStore[15].Axis[11].Pos12.Position := 0.0;
   AxisStore[15].Axis[11].Pos12.Speed := 0;
   AxisStore[15].Axis[11].Pos12.Reached := FALSE;
   AxisStore[15].Axis[11].Pos13.Position := 0.0;
   AxisStore[15].Axis[11].Pos13.Speed := 0;
   AxisStore[15].Axis[11].Pos13.Reached := FALSE;
   AxisStore[15].Axis[11].Pos14.Position := 0.0;
   AxisStore[15].Axis[11].Pos14.Speed := 0;
   AxisStore[15].Axis[11].Pos14.Reached := FALSE;
   AxisStore[15].Axis[11].Pos15.Position := 0.0;
   AxisStore[15].Axis[11].Pos15.Speed := 0;
   AxisStore[15].Axis[11].Pos15.Reached := FALSE;
   AxisStore[15].Axis[11].Pos16.Position := 0.0;
   AxisStore[15].Axis[11].Pos16.Speed := 0;
   AxisStore[15].Axis[11].Pos16.Reached := FALSE;
   AxisStore[15].Axis[11].Pos17.Position := 0.0;
   AxisStore[15].Axis[11].Pos17.Speed := 0;
   AxisStore[15].Axis[11].Pos17.Reached := FALSE;
   AxisStore[15].Axis[11].Pos18.Position := 0.0;
   AxisStore[15].Axis[11].Pos18.Speed := 0;
   AxisStore[15].Axis[11].Pos18.Reached := FALSE;
   AxisStore[15].Axis[11].Pos19.Position := 0.0;
   AxisStore[15].Axis[11].Pos19.Speed := 0;
   AxisStore[15].Axis[11].Pos19.Reached := FALSE;
   AxisStore[15].Axis[11].Pos20.Position := 0.0;
   AxisStore[15].Axis[11].Pos20.Speed := 0;
   AxisStore[15].Axis[11].Pos20.Reached := FALSE;
   AxisStore[15].Axis[11].Pos21.Position := 0.0;
   AxisStore[15].Axis[11].Pos21.Speed := 0;
   AxisStore[15].Axis[11].Pos21.Reached := FALSE;
   AxisStore[15].Axis[11].Pos22.Position := 0.0;
   AxisStore[15].Axis[11].Pos22.Speed := 0;
   AxisStore[15].Axis[11].Pos22.Reached := FALSE;
   AxisStore[15].Axis[11].Pos23.Position := 0.0;
   AxisStore[15].Axis[11].Pos23.Speed := 0;
   AxisStore[15].Axis[11].Pos23.Reached := FALSE;
   AxisStore[15].Axis[11].Pos24.Position := 0.0;
   AxisStore[15].Axis[11].Pos24.Speed := 0;
   AxisStore[15].Axis[11].Pos24.Reached := FALSE;
   AxisStore[15].Axis[11].Pos25.Position := 0.0;
   AxisStore[15].Axis[11].Pos25.Speed := 0;
   AxisStore[15].Axis[11].Pos25.Reached := FALSE;
   AxisStore[15].Axis[11].Pos26.Position := 0.0;
   AxisStore[15].Axis[11].Pos26.Speed := 0;
   AxisStore[15].Axis[11].Pos26.Reached := FALSE;
   AxisStore[15].Axis[11].Pos27.Position := 0.0;
   AxisStore[15].Axis[11].Pos27.Speed := 0;
   AxisStore[15].Axis[11].Pos27.Reached := FALSE;
   AxisStore[15].Axis[11].Pos28.Position := 0.0;
   AxisStore[15].Axis[11].Pos28.Speed := 0;
   AxisStore[15].Axis[11].Pos28.Reached := FALSE;
   AxisStore[15].Axis[11].Pos29.Position := 0.0;
   AxisStore[15].Axis[11].Pos29.Speed := 0;
   AxisStore[15].Axis[11].Pos29.Reached := FALSE;
   AxisStore[15].Axis[11].Pos30.Position := 0.0;
   AxisStore[15].Axis[11].Pos30.Speed := 0;
   AxisStore[15].Axis[11].Pos30.Reached := FALSE;
   AxisStore[15].Axis[12].Pos1.Position := 0.0;
   AxisStore[15].Axis[12].Pos1.Speed := 0;
   AxisStore[15].Axis[12].Pos1.Reached := FALSE;
   AxisStore[15].Axis[12].Pos2.Position := 0.0;
   AxisStore[15].Axis[12].Pos2.Speed := 0;
   AxisStore[15].Axis[12].Pos2.Reached := FALSE;
   AxisStore[15].Axis[12].Pos3.Position := 0.0;
   AxisStore[15].Axis[12].Pos3.Speed := 0;
   AxisStore[15].Axis[12].Pos3.Reached := FALSE;
   AxisStore[15].Axis[12].Pos4.Position := 0.0;
   AxisStore[15].Axis[12].Pos4.Speed := 0;
   AxisStore[15].Axis[12].Pos4.Reached := FALSE;
   AxisStore[15].Axis[12].Pos5.Position := 0.0;
   AxisStore[15].Axis[12].Pos5.Speed := 0;
   AxisStore[15].Axis[12].Pos5.Reached := FALSE;
   AxisStore[15].Axis[12].Pos6.Position := 0.0;
   AxisStore[15].Axis[12].Pos6.Speed := 0;
   AxisStore[15].Axis[12].Pos6.Reached := FALSE;
   AxisStore[15].Axis[12].Pos7.Position := 0.0;
   AxisStore[15].Axis[12].Pos7.Speed := 0;
   AxisStore[15].Axis[12].Pos7.Reached := FALSE;
   AxisStore[15].Axis[12].Pos8.Position := 0.0;
   AxisStore[15].Axis[12].Pos8.Speed := 0;
   AxisStore[15].Axis[12].Pos8.Reached := FALSE;
   AxisStore[15].Axis[12].Pos9.Position := 0.0;
   AxisStore[15].Axis[12].Pos9.Speed := 0;
   AxisStore[15].Axis[12].Pos9.Reached := FALSE;
   AxisStore[15].Axis[12].Pos10.Position := 0.0;
   AxisStore[15].Axis[12].Pos10.Speed := 0;
   AxisStore[15].Axis[12].Pos10.Reached := FALSE;
   AxisStore[15].Axis[12].Pos11.Position := 0.0;
   AxisStore[15].Axis[12].Pos11.Speed := 0;
   AxisStore[15].Axis[12].Pos11.Reached := FALSE;
   AxisStore[15].Axis[12].Pos12.Position := 0.0;
   AxisStore[15].Axis[12].Pos12.Speed := 0;
   AxisStore[15].Axis[12].Pos12.Reached := FALSE;
   AxisStore[15].Axis[12].Pos13.Position := 0.0;
   AxisStore[15].Axis[12].Pos13.Speed := 0;
   AxisStore[15].Axis[12].Pos13.Reached := FALSE;
   AxisStore[15].Axis[12].Pos14.Position := 0.0;
   AxisStore[15].Axis[12].Pos14.Speed := 0;
   AxisStore[15].Axis[12].Pos14.Reached := FALSE;
   AxisStore[15].Axis[12].Pos15.Position := 0.0;
   AxisStore[15].Axis[12].Pos15.Speed := 0;
   AxisStore[15].Axis[12].Pos15.Reached := FALSE;
   AxisStore[15].Axis[12].Pos16.Position := 0.0;
   AxisStore[15].Axis[12].Pos16.Speed := 0;
   AxisStore[15].Axis[12].Pos16.Reached := FALSE;
   AxisStore[15].Axis[12].Pos17.Position := 0.0;
   AxisStore[15].Axis[12].Pos17.Speed := 0;
   AxisStore[15].Axis[12].Pos17.Reached := FALSE;
   AxisStore[15].Axis[12].Pos18.Position := 0.0;
   AxisStore[15].Axis[12].Pos18.Speed := 0;
   AxisStore[15].Axis[12].Pos18.Reached := FALSE;
   AxisStore[15].Axis[12].Pos19.Position := 0.0;
   AxisStore[15].Axis[12].Pos19.Speed := 0;
   AxisStore[15].Axis[12].Pos19.Reached := FALSE;
   AxisStore[15].Axis[12].Pos20.Position := 0.0;
   AxisStore[15].Axis[12].Pos20.Speed := 0;
   AxisStore[15].Axis[12].Pos20.Reached := FALSE;
   AxisStore[15].Axis[12].Pos21.Position := 0.0;
   AxisStore[15].Axis[12].Pos21.Speed := 0;
   AxisStore[15].Axis[12].Pos21.Reached := FALSE;
   AxisStore[15].Axis[12].Pos22.Position := 0.0;
   AxisStore[15].Axis[12].Pos22.Speed := 0;
   AxisStore[15].Axis[12].Pos22.Reached := FALSE;
   AxisStore[15].Axis[12].Pos23.Position := 0.0;
   AxisStore[15].Axis[12].Pos23.Speed := 0;
   AxisStore[15].Axis[12].Pos23.Reached := FALSE;
   AxisStore[15].Axis[12].Pos24.Position := 0.0;
   AxisStore[15].Axis[12].Pos24.Speed := 0;
   AxisStore[15].Axis[12].Pos24.Reached := FALSE;
   AxisStore[15].Axis[12].Pos25.Position := 0.0;
   AxisStore[15].Axis[12].Pos25.Speed := 0;
   AxisStore[15].Axis[12].Pos25.Reached := FALSE;
   AxisStore[15].Axis[12].Pos26.Position := 0.0;
   AxisStore[15].Axis[12].Pos26.Speed := 0;
   AxisStore[15].Axis[12].Pos26.Reached := FALSE;
   AxisStore[15].Axis[12].Pos27.Position := 0.0;
   AxisStore[15].Axis[12].Pos27.Speed := 0;
   AxisStore[15].Axis[12].Pos27.Reached := FALSE;
   AxisStore[15].Axis[12].Pos28.Position := 0.0;
   AxisStore[15].Axis[12].Pos28.Speed := 0;
   AxisStore[15].Axis[12].Pos28.Reached := FALSE;
   AxisStore[15].Axis[12].Pos29.Position := 0.0;
   AxisStore[15].Axis[12].Pos29.Speed := 0;
   AxisStore[15].Axis[12].Pos29.Reached := FALSE;
   AxisStore[15].Axis[12].Pos30.Position := 0.0;
   AxisStore[15].Axis[12].Pos30.Speed := 0;
   AxisStore[15].Axis[12].Pos30.Reached := FALSE;
   AxisStore[15].Axis[13].Pos1.Position := 0.0;
   AxisStore[15].Axis[13].Pos1.Speed := 0;
   AxisStore[15].Axis[13].Pos1.Reached := FALSE;
   AxisStore[15].Axis[13].Pos2.Position := 0.0;
   AxisStore[15].Axis[13].Pos2.Speed := 0;
   AxisStore[15].Axis[13].Pos2.Reached := FALSE;
   AxisStore[15].Axis[13].Pos3.Position := 0.0;
   AxisStore[15].Axis[13].Pos3.Speed := 0;
   AxisStore[15].Axis[13].Pos3.Reached := FALSE;
   AxisStore[15].Axis[13].Pos4.Position := 0.0;
   AxisStore[15].Axis[13].Pos4.Speed := 0;
   AxisStore[15].Axis[13].Pos4.Reached := FALSE;
   AxisStore[15].Axis[13].Pos5.Position := 0.0;
   AxisStore[15].Axis[13].Pos5.Speed := 0;
   AxisStore[15].Axis[13].Pos5.Reached := FALSE;
   AxisStore[15].Axis[13].Pos6.Position := 0.0;
   AxisStore[15].Axis[13].Pos6.Speed := 0;
   AxisStore[15].Axis[13].Pos6.Reached := FALSE;
   AxisStore[15].Axis[13].Pos7.Position := 0.0;
   AxisStore[15].Axis[13].Pos7.Speed := 0;
   AxisStore[15].Axis[13].Pos7.Reached := FALSE;
   AxisStore[15].Axis[13].Pos8.Position := 0.0;
   AxisStore[15].Axis[13].Pos8.Speed := 0;
   AxisStore[15].Axis[13].Pos8.Reached := FALSE;
   AxisStore[15].Axis[13].Pos9.Position := 0.0;
   AxisStore[15].Axis[13].Pos9.Speed := 0;
   AxisStore[15].Axis[13].Pos9.Reached := FALSE;
   AxisStore[15].Axis[13].Pos10.Position := 0.0;
   AxisStore[15].Axis[13].Pos10.Speed := 0;
   AxisStore[15].Axis[13].Pos10.Reached := FALSE;
   AxisStore[15].Axis[13].Pos11.Position := 0.0;
   AxisStore[15].Axis[13].Pos11.Speed := 0;
   AxisStore[15].Axis[13].Pos11.Reached := FALSE;
   AxisStore[15].Axis[13].Pos12.Position := 0.0;
   AxisStore[15].Axis[13].Pos12.Speed := 0;
   AxisStore[15].Axis[13].Pos12.Reached := FALSE;
   AxisStore[15].Axis[13].Pos13.Position := 0.0;
   AxisStore[15].Axis[13].Pos13.Speed := 0;
   AxisStore[15].Axis[13].Pos13.Reached := FALSE;
   AxisStore[15].Axis[13].Pos14.Position := 0.0;
   AxisStore[15].Axis[13].Pos14.Speed := 0;
   AxisStore[15].Axis[13].Pos14.Reached := FALSE;
   AxisStore[15].Axis[13].Pos15.Position := 0.0;
   AxisStore[15].Axis[13].Pos15.Speed := 0;
   AxisStore[15].Axis[13].Pos15.Reached := FALSE;
   AxisStore[15].Axis[13].Pos16.Position := 0.0;
   AxisStore[15].Axis[13].Pos16.Speed := 0;
   AxisStore[15].Axis[13].Pos16.Reached := FALSE;
   AxisStore[15].Axis[13].Pos17.Position := 0.0;
   AxisStore[15].Axis[13].Pos17.Speed := 0;
   AxisStore[15].Axis[13].Pos17.Reached := FALSE;
   AxisStore[15].Axis[13].Pos18.Position := 0.0;
   AxisStore[15].Axis[13].Pos18.Speed := 0;
   AxisStore[15].Axis[13].Pos18.Reached := FALSE;
   AxisStore[15].Axis[13].Pos19.Position := 0.0;
   AxisStore[15].Axis[13].Pos19.Speed := 0;
   AxisStore[15].Axis[13].Pos19.Reached := FALSE;
   AxisStore[15].Axis[13].Pos20.Position := 0.0;
   AxisStore[15].Axis[13].Pos20.Speed := 0;
   AxisStore[15].Axis[13].Pos20.Reached := FALSE;
   AxisStore[15].Axis[13].Pos21.Position := 0.0;
   AxisStore[15].Axis[13].Pos21.Speed := 0;
   AxisStore[15].Axis[13].Pos21.Reached := FALSE;
   AxisStore[15].Axis[13].Pos22.Position := 0.0;
   AxisStore[15].Axis[13].Pos22.Speed := 0;
   AxisStore[15].Axis[13].Pos22.Reached := FALSE;
   AxisStore[15].Axis[13].Pos23.Position := 0.0;
   AxisStore[15].Axis[13].Pos23.Speed := 0;
   AxisStore[15].Axis[13].Pos23.Reached := FALSE;
   AxisStore[15].Axis[13].Pos24.Position := 0.0;
   AxisStore[15].Axis[13].Pos24.Speed := 0;
   AxisStore[15].Axis[13].Pos24.Reached := FALSE;
   AxisStore[15].Axis[13].Pos25.Position := 0.0;
   AxisStore[15].Axis[13].Pos25.Speed := 0;
   AxisStore[15].Axis[13].Pos25.Reached := FALSE;
   AxisStore[15].Axis[13].Pos26.Position := 0.0;
   AxisStore[15].Axis[13].Pos26.Speed := 0;
   AxisStore[15].Axis[13].Pos26.Reached := FALSE;
   AxisStore[15].Axis[13].Pos27.Position := 0.0;
   AxisStore[15].Axis[13].Pos27.Speed := 0;
   AxisStore[15].Axis[13].Pos27.Reached := FALSE;
   AxisStore[15].Axis[13].Pos28.Position := 0.0;
   AxisStore[15].Axis[13].Pos28.Speed := 0;
   AxisStore[15].Axis[13].Pos28.Reached := FALSE;
   AxisStore[15].Axis[13].Pos29.Position := 0.0;
   AxisStore[15].Axis[13].Pos29.Speed := 0;
   AxisStore[15].Axis[13].Pos29.Reached := FALSE;
   AxisStore[15].Axis[13].Pos30.Position := 0.0;
   AxisStore[15].Axis[13].Pos30.Speed := 0;
   AxisStore[15].Axis[13].Pos30.Reached := FALSE;
   AxisStore[15].Axis[14].Pos1.Position := 0.0;
   AxisStore[15].Axis[14].Pos1.Speed := 0;
   AxisStore[15].Axis[14].Pos1.Reached := FALSE;
   AxisStore[15].Axis[14].Pos2.Position := 0.0;
   AxisStore[15].Axis[14].Pos2.Speed := 0;
   AxisStore[15].Axis[14].Pos2.Reached := FALSE;
   AxisStore[15].Axis[14].Pos3.Position := 0.0;
   AxisStore[15].Axis[14].Pos3.Speed := 0;
   AxisStore[15].Axis[14].Pos3.Reached := FALSE;
   AxisStore[15].Axis[14].Pos4.Position := 0.0;
   AxisStore[15].Axis[14].Pos4.Speed := 0;
   AxisStore[15].Axis[14].Pos4.Reached := FALSE;
   AxisStore[15].Axis[14].Pos5.Position := 0.0;
   AxisStore[15].Axis[14].Pos5.Speed := 0;
   AxisStore[15].Axis[14].Pos5.Reached := FALSE;
   AxisStore[15].Axis[14].Pos6.Position := 0.0;
   AxisStore[15].Axis[14].Pos6.Speed := 0;
   AxisStore[15].Axis[14].Pos6.Reached := FALSE;
   AxisStore[15].Axis[14].Pos7.Position := 0.0;
   AxisStore[15].Axis[14].Pos7.Speed := 0;
   AxisStore[15].Axis[14].Pos7.Reached := FALSE;
   AxisStore[15].Axis[14].Pos8.Position := 0.0;
   AxisStore[15].Axis[14].Pos8.Speed := 0;
   AxisStore[15].Axis[14].Pos8.Reached := FALSE;
   AxisStore[15].Axis[14].Pos9.Position := 0.0;
   AxisStore[15].Axis[14].Pos9.Speed := 0;
   AxisStore[15].Axis[14].Pos9.Reached := FALSE;
   AxisStore[15].Axis[14].Pos10.Position := 0.0;
   AxisStore[15].Axis[14].Pos10.Speed := 0;
   AxisStore[15].Axis[14].Pos10.Reached := FALSE;
   AxisStore[15].Axis[14].Pos11.Position := 0.0;
   AxisStore[15].Axis[14].Pos11.Speed := 0;
   AxisStore[15].Axis[14].Pos11.Reached := FALSE;
   AxisStore[15].Axis[14].Pos12.Position := 0.0;
   AxisStore[15].Axis[14].Pos12.Speed := 0;
   AxisStore[15].Axis[14].Pos12.Reached := FALSE;
   AxisStore[15].Axis[14].Pos13.Position := 0.0;
   AxisStore[15].Axis[14].Pos13.Speed := 0;
   AxisStore[15].Axis[14].Pos13.Reached := FALSE;
   AxisStore[15].Axis[14].Pos14.Position := 0.0;
   AxisStore[15].Axis[14].Pos14.Speed := 0;
   AxisStore[15].Axis[14].Pos14.Reached := FALSE;
   AxisStore[15].Axis[14].Pos15.Position := 0.0;
   AxisStore[15].Axis[14].Pos15.Speed := 0;
   AxisStore[15].Axis[14].Pos15.Reached := FALSE;
   AxisStore[15].Axis[14].Pos16.Position := 0.0;
   AxisStore[15].Axis[14].Pos16.Speed := 0;
   AxisStore[15].Axis[14].Pos16.Reached := FALSE;
   AxisStore[15].Axis[14].Pos17.Position := 0.0;
   AxisStore[15].Axis[14].Pos17.Speed := 0;
   AxisStore[15].Axis[14].Pos17.Reached := FALSE;
   AxisStore[15].Axis[14].Pos18.Position := 0.0;
   AxisStore[15].Axis[14].Pos18.Speed := 0;
   AxisStore[15].Axis[14].Pos18.Reached := FALSE;
   AxisStore[15].Axis[14].Pos19.Position := 0.0;
   AxisStore[15].Axis[14].Pos19.Speed := 0;
   AxisStore[15].Axis[14].Pos19.Reached := FALSE;
   AxisStore[15].Axis[14].Pos20.Position := 0.0;
   AxisStore[15].Axis[14].Pos20.Speed := 0;
   AxisStore[15].Axis[14].Pos20.Reached := FALSE;
   AxisStore[15].Axis[14].Pos21.Position := 0.0;
   AxisStore[15].Axis[14].Pos21.Speed := 0;
   AxisStore[15].Axis[14].Pos21.Reached := FALSE;
   AxisStore[15].Axis[14].Pos22.Position := 0.0;
   AxisStore[15].Axis[14].Pos22.Speed := 0;
   AxisStore[15].Axis[14].Pos22.Reached := FALSE;
   AxisStore[15].Axis[14].Pos23.Position := 0.0;
   AxisStore[15].Axis[14].Pos23.Speed := 0;
   AxisStore[15].Axis[14].Pos23.Reached := FALSE;
   AxisStore[15].Axis[14].Pos24.Position := 0.0;
   AxisStore[15].Axis[14].Pos24.Speed := 0;
   AxisStore[15].Axis[14].Pos24.Reached := FALSE;
   AxisStore[15].Axis[14].Pos25.Position := 0.0;
   AxisStore[15].Axis[14].Pos25.Speed := 0;
   AxisStore[15].Axis[14].Pos25.Reached := FALSE;
   AxisStore[15].Axis[14].Pos26.Position := 0.0;
   AxisStore[15].Axis[14].Pos26.Speed := 0;
   AxisStore[15].Axis[14].Pos26.Reached := FALSE;
   AxisStore[15].Axis[14].Pos27.Position := 0.0;
   AxisStore[15].Axis[14].Pos27.Speed := 0;
   AxisStore[15].Axis[14].Pos27.Reached := FALSE;
   AxisStore[15].Axis[14].Pos28.Position := 0.0;
   AxisStore[15].Axis[14].Pos28.Speed := 0;
   AxisStore[15].Axis[14].Pos28.Reached := FALSE;
   AxisStore[15].Axis[14].Pos29.Position := 0.0;
   AxisStore[15].Axis[14].Pos29.Speed := 0;
   AxisStore[15].Axis[14].Pos29.Reached := FALSE;
   AxisStore[15].Axis[14].Pos30.Position := 0.0;
   AxisStore[15].Axis[14].Pos30.Speed := 0;
   AxisStore[15].Axis[14].Pos30.Reached := FALSE;
   AxisStore[15].Axis[15].Pos1.Position := 0.0;
   AxisStore[15].Axis[15].Pos1.Speed := 0;
   AxisStore[15].Axis[15].Pos1.Reached := FALSE;
   AxisStore[15].Axis[15].Pos2.Position := 0.0;
   AxisStore[15].Axis[15].Pos2.Speed := 0;
   AxisStore[15].Axis[15].Pos2.Reached := FALSE;
   AxisStore[15].Axis[15].Pos3.Position := 0.0;
   AxisStore[15].Axis[15].Pos3.Speed := 0;
   AxisStore[15].Axis[15].Pos3.Reached := FALSE;
   AxisStore[15].Axis[15].Pos4.Position := 0.0;
   AxisStore[15].Axis[15].Pos4.Speed := 0;
   AxisStore[15].Axis[15].Pos4.Reached := FALSE;
   AxisStore[15].Axis[15].Pos5.Position := 0.0;
   AxisStore[15].Axis[15].Pos5.Speed := 0;
   AxisStore[15].Axis[15].Pos5.Reached := FALSE;
   AxisStore[15].Axis[15].Pos6.Position := 0.0;
   AxisStore[15].Axis[15].Pos6.Speed := 0;
   AxisStore[15].Axis[15].Pos6.Reached := FALSE;
   AxisStore[15].Axis[15].Pos7.Position := 0.0;
   AxisStore[15].Axis[15].Pos7.Speed := 0;
   AxisStore[15].Axis[15].Pos7.Reached := FALSE;
   AxisStore[15].Axis[15].Pos8.Position := 0.0;
   AxisStore[15].Axis[15].Pos8.Speed := 0;
   AxisStore[15].Axis[15].Pos8.Reached := FALSE;
   AxisStore[15].Axis[15].Pos9.Position := 0.0;
   AxisStore[15].Axis[15].Pos9.Speed := 0;
   AxisStore[15].Axis[15].Pos9.Reached := FALSE;
   AxisStore[15].Axis[15].Pos10.Position := 0.0;
   AxisStore[15].Axis[15].Pos10.Speed := 0;
   AxisStore[15].Axis[15].Pos10.Reached := FALSE;
   AxisStore[15].Axis[15].Pos11.Position := 0.0;
   AxisStore[15].Axis[15].Pos11.Speed := 0;
   AxisStore[15].Axis[15].Pos11.Reached := FALSE;
   AxisStore[15].Axis[15].Pos12.Position := 0.0;
   AxisStore[15].Axis[15].Pos12.Speed := 0;
   AxisStore[15].Axis[15].Pos12.Reached := FALSE;
   AxisStore[15].Axis[15].Pos13.Position := 0.0;
   AxisStore[15].Axis[15].Pos13.Speed := 0;
   AxisStore[15].Axis[15].Pos13.Reached := FALSE;
   AxisStore[15].Axis[15].Pos14.Position := 0.0;
   AxisStore[15].Axis[15].Pos14.Speed := 0;
   AxisStore[15].Axis[15].Pos14.Reached := FALSE;
   AxisStore[15].Axis[15].Pos15.Position := 0.0;
   AxisStore[15].Axis[15].Pos15.Speed := 0;
   AxisStore[15].Axis[15].Pos15.Reached := FALSE;
   AxisStore[15].Axis[15].Pos16.Position := 0.0;
   AxisStore[15].Axis[15].Pos16.Speed := 0;
   AxisStore[15].Axis[15].Pos16.Reached := FALSE;
   AxisStore[15].Axis[15].Pos17.Position := 0.0;
   AxisStore[15].Axis[15].Pos17.Speed := 0;
   AxisStore[15].Axis[15].Pos17.Reached := FALSE;
   AxisStore[15].Axis[15].Pos18.Position := 0.0;
   AxisStore[15].Axis[15].Pos18.Speed := 0;
   AxisStore[15].Axis[15].Pos18.Reached := FALSE;
   AxisStore[15].Axis[15].Pos19.Position := 0.0;
   AxisStore[15].Axis[15].Pos19.Speed := 0;
   AxisStore[15].Axis[15].Pos19.Reached := FALSE;
   AxisStore[15].Axis[15].Pos20.Position := 0.0;
   AxisStore[15].Axis[15].Pos20.Speed := 0;
   AxisStore[15].Axis[15].Pos20.Reached := FALSE;
   AxisStore[15].Axis[15].Pos21.Position := 0.0;
   AxisStore[15].Axis[15].Pos21.Speed := 0;
   AxisStore[15].Axis[15].Pos21.Reached := FALSE;
   AxisStore[15].Axis[15].Pos22.Position := 0.0;
   AxisStore[15].Axis[15].Pos22.Speed := 0;
   AxisStore[15].Axis[15].Pos22.Reached := FALSE;
   AxisStore[15].Axis[15].Pos23.Position := 0.0;
   AxisStore[15].Axis[15].Pos23.Speed := 0;
   AxisStore[15].Axis[15].Pos23.Reached := FALSE;
   AxisStore[15].Axis[15].Pos24.Position := 0.0;
   AxisStore[15].Axis[15].Pos24.Speed := 0;
   AxisStore[15].Axis[15].Pos24.Reached := FALSE;
   AxisStore[15].Axis[15].Pos25.Position := 0.0;
   AxisStore[15].Axis[15].Pos25.Speed := 0;
   AxisStore[15].Axis[15].Pos25.Reached := FALSE;
   AxisStore[15].Axis[15].Pos26.Position := 0.0;
   AxisStore[15].Axis[15].Pos26.Speed := 0;
   AxisStore[15].Axis[15].Pos26.Reached := FALSE;
   AxisStore[15].Axis[15].Pos27.Position := 0.0;
   AxisStore[15].Axis[15].Pos27.Speed := 0;
   AxisStore[15].Axis[15].Pos27.Reached := FALSE;
   AxisStore[15].Axis[15].Pos28.Position := 0.0;
   AxisStore[15].Axis[15].Pos28.Speed := 0;
   AxisStore[15].Axis[15].Pos28.Reached := FALSE;
   AxisStore[15].Axis[15].Pos29.Position := 0.0;
   AxisStore[15].Axis[15].Pos29.Speed := 0;
   AxisStore[15].Axis[15].Pos29.Reached := FALSE;
   AxisStore[15].Axis[15].Pos30.Position := 0.0;
   AxisStore[15].Axis[15].Pos30.Speed := 0;
   AxisStore[15].Axis[15].Pos30.Reached := FALSE;

END_DATA_BLOCK

DATA_BLOCK "ST10_RecipeActiveDB"
{ S7_Optimized_Access := 'FALSE' }
VERSION : 0.1
   STRUCT 
      Recipe : Struct
         RecipeTag : String[50];
         RecordName : String[50];
         PreConfigType : String[50];
         Pulse : Bool;
         Trigger : Bool;
         PosEdg : Bool;
         Alarm : Bool;
         Ret : Bool;
         Equal : Bool;
         Pls : Bool;
         "time" : Int;
         Spare : Array[0..38] of Byte;
         DataRecord_TransferStatus : Int;
      END_STRUCT;
      ParameterElement : Struct
         TypeName : String[50];
         TypeID : Int;
         FixtureID : Array[0..5] of Int;
         FestoAxis { S7_SetPoint := 'False'} : "RecipeAxis";
         PressRgramNo { S7_SetPoint := 'True'} : Array[0..60] of DInt;
         ProcessParameter : "MEStoPLC_RecipeData_OP220";
      END_STRUCT;
   END_STRUCT;


BEGIN

END_DATA_BLOCK

DATA_BLOCK "ST10_RecipeDB"
{ S7_Optimized_Access := 'FALSE' }
VERSION : 0.1
   STRUCT 
      Recipe : Struct
         RecipeTag : String[50];   // System Defined=
         RecordName : String[50];   // 配方名称ID
         PreConfigType : String[50];   // 数据记录名称
         Pulse : Bool;   // 待切换数据记录名称
         Trigger : Bool;
         PosEdg : Bool;   // 配方切换触发
         Alarm : Bool;
         Ret : Bool;
         Equal : Bool;
         Pls : Bool;   // 换型OK标志位
         "time" : Int;
         Spare : Array[0..38] of Byte;
         DataRecord_TransferStatus : Int;   // 数据记录传送状态
      END_STRUCT;
      ParameterElement : Struct
         TypeName : String[50];   // System Defined=
         TypeID : USInt;   // System define= product type for parameters of servo ,press and so on
         FixtureID : Array[1..16] of Byte;
         A1_TableFixtureCode : Array[0..10] of String[128];
         A2_TableFixtureCode : Array[0..10] of String[128];
         A1RingUnloadingFixtureCode : String[128];
         E1LoadingNGFixtureCode : String[128];
         ShaftScanFixtureCode : String[128];
         B1PressFixtureCode : String[128];
         CGlueFixtureCode : String[128];
         B1PressCylFixtureCode : String[128];
         A2RingUnloadingFixtureCode : String[128];
         E2UnloadingNGFixtureCode : String[128];
         B2PressFixtureCode : String[128];
         CGlueNGFixtureCode : String[128];
         B2PressCylFixtureCode : String[128];
         R1GripperFixtureCode : Array[0..6] of String[128];
         R2GripperFixtureCode : Array[0..6] of String[128];
         R3GripperFixtureCode : Array[0..6] of String[128];
         B1PressProgram : Int;
         B2PressProgram : Int;
         CGlueShaftIV3Program_1 : Word;
         CGlueShaftIV3Program_2 : Word;
         CGlueShaftIV3Program_3 : Word;
         CGlueShaftIV3Program_4 : Word;
         CGlueMagnetIV3Program : Word;
         CGlueProgram : Int;
      END_STRUCT;
   END_STRUCT;


BEGIN
   Recipe.RecipeTag := 'RecipeST10';
   Recipe.RecordName := 'Product_1';
   Recipe.PreConfigType := 'Product_1';
   Recipe.Pulse := FALSE;
   Recipe.Trigger := FALSE;
   Recipe.PosEdg := FALSE;
   Recipe.Alarm := FALSE;
   Recipe.Ret := FALSE;
   Recipe.Equal := TRUE;
   Recipe.Pls := FALSE;
   Recipe."time" := 0;
   Recipe.Spare[0] := 16#00;
   Recipe.Spare[1] := 16#00;
   Recipe.Spare[2] := 16#00;
   Recipe.Spare[3] := 16#00;
   Recipe.Spare[4] := 16#00;
   Recipe.Spare[5] := 16#00;
   Recipe.Spare[6] := 16#00;
   Recipe.Spare[7] := 16#00;
   Recipe.Spare[8] := 16#00;
   Recipe.Spare[9] := 16#00;
   Recipe.Spare[10] := 16#00;
   Recipe.Spare[11] := 16#00;
   Recipe.Spare[12] := 16#00;
   Recipe.Spare[13] := 16#00;
   Recipe.Spare[14] := 16#00;
   Recipe.Spare[15] := 16#00;
   Recipe.Spare[16] := 16#00;
   Recipe.Spare[17] := 16#00;
   Recipe.Spare[18] := 16#00;
   Recipe.Spare[19] := 16#00;
   Recipe.Spare[20] := 16#00;
   Recipe.Spare[21] := 16#00;
   Recipe.Spare[22] := 16#00;
   Recipe.Spare[23] := 16#00;
   Recipe.Spare[24] := 16#00;
   Recipe.Spare[25] := 16#00;
   Recipe.Spare[26] := 16#00;
   Recipe.Spare[27] := 16#00;
   Recipe.Spare[28] := 16#00;
   Recipe.Spare[29] := 16#00;
   Recipe.Spare[30] := 16#00;
   Recipe.Spare[31] := 16#00;
   Recipe.Spare[32] := 16#00;
   Recipe.Spare[33] := 16#00;
   Recipe.Spare[34] := 16#00;
   Recipe.Spare[35] := 16#00;
   Recipe.Spare[36] := 16#00;
   Recipe.Spare[37] := 16#00;
   Recipe.Spare[38] := 16#00;
   Recipe.DataRecord_TransferStatus := 0;
   ParameterElement.TypeName := 'Product_1';
   ParameterElement.TypeID := 1;
   ParameterElement.FixtureID[1] := 16#00;
   ParameterElement.FixtureID[2] := 16#00;
   ParameterElement.FixtureID[3] := 16#00;
   ParameterElement.FixtureID[4] := 16#00;
   ParameterElement.FixtureID[5] := 16#00;
   ParameterElement.FixtureID[6] := 16#00;
   ParameterElement.FixtureID[7] := 16#00;
   ParameterElement.FixtureID[8] := 16#00;
   ParameterElement.FixtureID[9] := 16#00;
   ParameterElement.FixtureID[10] := 16#00;
   ParameterElement.FixtureID[11] := 16#00;
   ParameterElement.FixtureID[12] := 16#00;
   ParameterElement.FixtureID[13] := 16#00;
   ParameterElement.FixtureID[14] := 16#00;
   ParameterElement.FixtureID[15] := 16#00;
   ParameterElement.FixtureID[16] := 16#00;
   ParameterElement.A1_TableFixtureCode[0] := '';
   ParameterElement.A1_TableFixtureCode[1] := 'SZ23055-OP010-E-Compressor-ring1 Loading tooling-1';
   ParameterElement.A1_TableFixtureCode[2] := 'SZ23055-OP010-E-Compressor-ring1 Loading tooling-2';
   ParameterElement.A1_TableFixtureCode[3] := 'SZ23055-OP010-E-Compressor-ring1 Loading tooling-3';
   ParameterElement.A1_TableFixtureCode[4] := 'SZ23055-OP010-E-Compressor-ring1 Loading tooling-4';
   ParameterElement.A1_TableFixtureCode[5] := 'SZ23055-OP010-E-Compressor-ring1 Loading tooling-5';
   ParameterElement.A1_TableFixtureCode[6] := 'SZ23055-OP010-E-Compressor-ring1 Loading tooling-6';
   ParameterElement.A1_TableFixtureCode[7] := 'SZ23055-OP010-E-Compressor-ring1 Loading tooling-7';
   ParameterElement.A1_TableFixtureCode[8] := 'SZ23055-OP010-E-Compressor-ring1 Loading tooling-8';
   ParameterElement.A1_TableFixtureCode[9] := '';
   ParameterElement.A1_TableFixtureCode[10] := '';
   ParameterElement.A2_TableFixtureCode[0] := '';
   ParameterElement.A2_TableFixtureCode[1] := 'SZ23055-OP010-E-Compressor-ring2 Loading tooling-1';
   ParameterElement.A2_TableFixtureCode[2] := 'SZ23055-OP010-E-Compressor-ring2 Loading tooling-2';
   ParameterElement.A2_TableFixtureCode[3] := 'SZ23055-OP010-E-Compressor-ring2 Loading tooling-3';
   ParameterElement.A2_TableFixtureCode[4] := 'SZ23055-OP010-E-Compressor-ring2 Loading tooling-4';
   ParameterElement.A2_TableFixtureCode[5] := 'SZ23055-OP010-E-Compressor-ring2 Loading tooling-5';
   ParameterElement.A2_TableFixtureCode[6] := 'SZ23055-OP010-E-Compressor-ring2 Loading tooling-6';
   ParameterElement.A2_TableFixtureCode[7] := 'SZ23055-OP010-E-Compressor-ring2 Loading tooling-7';
   ParameterElement.A2_TableFixtureCode[8] := 'SZ23055-OP010-E-Compressor-ring2 Loading tooling-8';
   ParameterElement.A2_TableFixtureCode[9] := '';
   ParameterElement.A2_TableFixtureCode[10] := '';
   ParameterElement.A1RingUnloadingFixtureCode := 'F2';
   ParameterElement.E1LoadingNGFixtureCode := 'SZ23055-OP010-E-Compressor-Left NG tooling-1';
   ParameterElement.ShaftScanFixtureCode := 'SZ23055-OP010-E-Compressor-shaft Rotating scanning tooling-1';
   ParameterElement.B1PressFixtureCode := 'SZ23055-OP010-E-Compressor-ring1 Below Positioning fixture -1';
   ParameterElement.CGlueFixtureCode := 'SZ23055-OP010-E-Compressor-Point adhesive tooling-1';
   ParameterElement.B1PressCylFixtureCode := 'SZ23055-OP010-E-Compressor-ring1 Upper pressing fixture-1';
   ParameterElement.A2RingUnloadingFixtureCode := 'F12';
   ParameterElement.E2UnloadingNGFixtureCode := 'SZ23055-OP010-E-Compressor-Right NG tooling-1';
   ParameterElement.B2PressFixtureCode := 'SZ23055-OP010-E-Compressor-ring2 Below Positioning fixture -1';
   ParameterElement.CGlueNGFixtureCode := 'SZ23055-OP010-E-Compressor-NG middle shift tooling-1';
   ParameterElement.B2PressCylFixtureCode := 'SZ23055-OP010-E-Compressor-ring2 Upper pressing fixture-1';
   ParameterElement.R1GripperFixtureCode[0] := '';
   ParameterElement.R1GripperFixtureCode[1] := 'SZ23055-OP010-E-Compressor-robot1 ring1 Left clamping jaw tooling-1';
   ParameterElement.R1GripperFixtureCode[2] := 'SZ23055-OP010-E-Compressor-robot1 ring1 Right clamping jaw tooling-2';
   ParameterElement.R1GripperFixtureCode[3] := 'SZ23055-OP010-E-Compressor-robot1 shaft Left clamping jaw tooling-1';
   ParameterElement.R1GripperFixtureCode[4] := 'SZ23055-OP010-E-Compressor-robot1 shaft Right clamping jaw tooling-2';
   ParameterElement.R1GripperFixtureCode[5] := '';
   ParameterElement.R1GripperFixtureCode[6] := '';
   ParameterElement.R2GripperFixtureCode[0] := '';
   ParameterElement.R2GripperFixtureCode[1] := 'SZ23055-OP010-E-Compressor-robot2 shaft Right clamping jaw tooling-2';
   ParameterElement.R2GripperFixtureCode[2] := 'SZ23055-OP010-E-Compressor-robot2 shaft Left clamping jaw tooling-1';
   ParameterElement.R2GripperFixtureCode[3] := 'SZ23055-OP010-E-Compressor-robot2 magnet Left clamping jaw tooling-1';
   ParameterElement.R2GripperFixtureCode[4] := 'SZ23055-OP010-E-Compressor-robot2 magnet Right clamping jaw tooling-2';
   ParameterElement.R2GripperFixtureCode[5] := '';
   ParameterElement.R2GripperFixtureCode[6] := '';
   ParameterElement.R3GripperFixtureCode[0] := '';
   ParameterElement.R3GripperFixtureCode[1] := 'SZ23055-OP010-E-Compressor-robot3 ring2 Right clamping jaw tooling-2';
   ParameterElement.R3GripperFixtureCode[2] := 'SZ23055-OP010-E-Compressor-robot3 ring2 Left clamping jaw tooling-1';
   ParameterElement.R3GripperFixtureCode[3] := 'SZ23055-OP010-E-Compressor-robot3 shaft Left clamping jaw tooling-1';
   ParameterElement.R3GripperFixtureCode[4] := 'SZ23055-OP010-E-Compressor-robot3 shaft Right clamping jaw tooling-2';
   ParameterElement.R3GripperFixtureCode[5] := '';
   ParameterElement.R3GripperFixtureCode[6] := '';
   ParameterElement.B1PressProgram := 1;
   ParameterElement.B2PressProgram := 1;
   ParameterElement.CGlueShaftIV3Program_1 := 16#0001;
   ParameterElement.CGlueShaftIV3Program_2 := 16#0002;
   ParameterElement.CGlueShaftIV3Program_3 := 16#0003;
   ParameterElement.CGlueShaftIV3Program_4 := 16#0004;
   ParameterElement.CGlueMagnetIV3Program := 16#0001;
   ParameterElement.CGlueProgram := 1;

END_DATA_BLOCK

DATA_BLOCK "ST10_RecipeDB_HMI"
{ S7_Optimized_Access := 'FALSE' }
VERSION : 0.1
   STRUCT 
      Recipe : Struct
         RecipeTag : String[50];   // System Defined=
         RecordName : String[50];   // 配方名称ID
         PreConfigType : String[50];   // 数据记录名称
         Pulse : Bool;   // 待切换数据记录名称
         Trigger : Bool;
         PosEdg : Bool;   // 配方切换触发
         Alarm : Bool;
         Ret : Bool;
         Equal : Bool;
         Pls : Bool;   // 换型OK标志位
         "time" : Int;
         Spare : Array[0..38] of Byte;
         DataRecord_TransferStatus : Int;   // 数据记录传送状态
      END_STRUCT;
      ParameterElement : Struct
         TypeName : String[50];   // System Defined=
         TypeID : USInt;   // System define= product type for parameters of servo ,press and so on
         FixtureID : Array[1..16] of Byte;
         A1_TableFixtureCode : Array[0..10] of String[128];
         A2_TableFixtureCode : Array[0..10] of String[128];
         A1RingUnloadingFixtureCode : String[128];
         E1LoadingNGFixtureCode : String[128];
         ShaftScanFixtureCode : String[128];
         B1PressFixtureCode : String[128];
         CGlueFixtureCode : String[128];
         B1PressCylFixtureCode : String[128];
         A2RingUnloadingFixtureCode : String[128];
         E2UnloadingNGFixtureCode : String[128];
         B2PressFixtureCode : String[128];
         CGlueNGFixtureCode : String[128];
         B2PressCylFixtureCode : String[128];
         R1GripperFixtureCode : Array[0..6] of String[128];
         R2GripperFixtureCode : Array[0..6] of String[128];
         R3GripperFixtureCode : Array[0..6] of String[128];
         B1PressProgram : Int;
         B2PressProgram : Int;
         CGlueShaftIV3Program_1 : Word;
         CGlueShaftIV3Program_2 : Word;
         CGlueShaftIV3Program_3 : Word;
         CGlueShaftIV3Program_4 : Word;
         CGlueMagnetIV3Program : Word;
         CGlueProgram : Int;
      END_STRUCT;
   END_STRUCT;


BEGIN
   Recipe.RecipeTag := 'RecipeST10';
   Recipe.RecordName := 'Product_1';
   Recipe.PreConfigType := 'Product_1';
   Recipe.Pulse := FALSE;
   Recipe.Trigger := FALSE;
   Recipe.PosEdg := TRUE;
   Recipe.Alarm := FALSE;
   Recipe.Ret := FALSE;
   Recipe.Equal := TRUE;
   Recipe.Pls := FALSE;
   Recipe."time" := 0;
   Recipe.Spare[0] := 16#00;
   Recipe.Spare[1] := 16#00;
   Recipe.Spare[2] := 16#00;
   Recipe.Spare[3] := 16#00;
   Recipe.Spare[4] := 16#00;
   Recipe.Spare[5] := 16#00;
   Recipe.Spare[6] := 16#00;
   Recipe.Spare[7] := 16#00;
   Recipe.Spare[8] := 16#00;
   Recipe.Spare[9] := 16#00;
   Recipe.Spare[10] := 16#00;
   Recipe.Spare[11] := 16#00;
   Recipe.Spare[12] := 16#00;
   Recipe.Spare[13] := 16#00;
   Recipe.Spare[14] := 16#00;
   Recipe.Spare[15] := 16#00;
   Recipe.Spare[16] := 16#00;
   Recipe.Spare[17] := 16#00;
   Recipe.Spare[18] := 16#00;
   Recipe.Spare[19] := 16#00;
   Recipe.Spare[20] := 16#00;
   Recipe.Spare[21] := 16#00;
   Recipe.Spare[22] := 16#00;
   Recipe.Spare[23] := 16#00;
   Recipe.Spare[24] := 16#00;
   Recipe.Spare[25] := 16#00;
   Recipe.Spare[26] := 16#00;
   Recipe.Spare[27] := 16#00;
   Recipe.Spare[28] := 16#00;
   Recipe.Spare[29] := 16#00;
   Recipe.Spare[30] := 16#00;
   Recipe.Spare[31] := 16#00;
   Recipe.Spare[32] := 16#00;
   Recipe.Spare[33] := 16#00;
   Recipe.Spare[34] := 16#00;
   Recipe.Spare[35] := 16#00;
   Recipe.Spare[36] := 16#00;
   Recipe.Spare[37] := 16#00;
   Recipe.Spare[38] := 16#00;
   Recipe.DataRecord_TransferStatus := 0;
   ParameterElement.TypeName := 'Product_1';
   ParameterElement.TypeID := 1;
   ParameterElement.FixtureID[1] := 16#00;
   ParameterElement.FixtureID[2] := 16#00;
   ParameterElement.FixtureID[3] := 16#00;
   ParameterElement.FixtureID[4] := 16#00;
   ParameterElement.FixtureID[5] := 16#00;
   ParameterElement.FixtureID[6] := 16#00;
   ParameterElement.FixtureID[7] := 16#00;
   ParameterElement.FixtureID[8] := 16#00;
   ParameterElement.FixtureID[9] := 16#00;
   ParameterElement.FixtureID[10] := 16#00;
   ParameterElement.FixtureID[11] := 16#00;
   ParameterElement.FixtureID[12] := 16#00;
   ParameterElement.FixtureID[13] := 16#00;
   ParameterElement.FixtureID[14] := 16#00;
   ParameterElement.FixtureID[15] := 16#00;
   ParameterElement.FixtureID[16] := 16#00;
   ParameterElement.A1_TableFixtureCode[0] := '';
   ParameterElement.A1_TableFixtureCode[1] := 'SZ23055-OP010-E-Compressor-ring1 Loading tooling-1';
   ParameterElement.A1_TableFixtureCode[2] := 'SZ23055-OP010-E-Compressor-ring1 Loading tooling-2';
   ParameterElement.A1_TableFixtureCode[3] := 'SZ23055-OP010-E-Compressor-ring1 Loading tooling-3';
   ParameterElement.A1_TableFixtureCode[4] := 'SZ23055-OP010-E-Compressor-ring1 Loading tooling-4';
   ParameterElement.A1_TableFixtureCode[5] := 'SZ23055-OP010-E-Compressor-ring1 Loading tooling-5';
   ParameterElement.A1_TableFixtureCode[6] := 'SZ23055-OP010-E-Compressor-ring1 Loading tooling-6';
   ParameterElement.A1_TableFixtureCode[7] := 'SZ23055-OP010-E-Compressor-ring1 Loading tooling-7';
   ParameterElement.A1_TableFixtureCode[8] := 'SZ23055-OP010-E-Compressor-ring1 Loading tooling-8';
   ParameterElement.A1_TableFixtureCode[9] := '';
   ParameterElement.A1_TableFixtureCode[10] := '';
   ParameterElement.A2_TableFixtureCode[0] := '';
   ParameterElement.A2_TableFixtureCode[1] := 'SZ23055-OP010-E-Compressor-ring2 Loading tooling-1';
   ParameterElement.A2_TableFixtureCode[2] := 'SZ23055-OP010-E-Compressor-ring2 Loading tooling-2';
   ParameterElement.A2_TableFixtureCode[3] := 'SZ23055-OP010-E-Compressor-ring2 Loading tooling-3';
   ParameterElement.A2_TableFixtureCode[4] := 'SZ23055-OP010-E-Compressor-ring2 Loading tooling-4';
   ParameterElement.A2_TableFixtureCode[5] := 'SZ23055-OP010-E-Compressor-ring2 Loading tooling-5';
   ParameterElement.A2_TableFixtureCode[6] := 'SZ23055-OP010-E-Compressor-ring2 Loading tooling-6';
   ParameterElement.A2_TableFixtureCode[7] := 'SZ23055-OP010-E-Compressor-ring2 Loading tooling-7';
   ParameterElement.A2_TableFixtureCode[8] := 'SZ23055-OP010-E-Compressor-ring2 Loading tooling-8';
   ParameterElement.A2_TableFixtureCode[9] := '';
   ParameterElement.A2_TableFixtureCode[10] := '';
   ParameterElement.A1RingUnloadingFixtureCode := 'F2';
   ParameterElement.E1LoadingNGFixtureCode := 'SZ23055-OP010-E-Compressor-Left NG tooling-1';
   ParameterElement.ShaftScanFixtureCode := 'SZ23055-OP010-E-Compressor-shaft Rotating scanning tooling-1';
   ParameterElement.B1PressFixtureCode := 'SZ23055-OP010-E-Compressor-ring1 Below Positioning fixture -1';
   ParameterElement.CGlueFixtureCode := 'SZ23055-OP010-E-Compressor-Point adhesive tooling-1';
   ParameterElement.B1PressCylFixtureCode := 'SZ23055-OP010-E-Compressor-ring1 Upper pressing fixture-1';
   ParameterElement.A2RingUnloadingFixtureCode := 'F12';
   ParameterElement.E2UnloadingNGFixtureCode := 'SZ23055-OP010-E-Compressor-Right NG tooling-1';
   ParameterElement.B2PressFixtureCode := 'SZ23055-OP010-E-Compressor-ring2 Below Positioning fixture -1';
   ParameterElement.CGlueNGFixtureCode := 'SZ23055-OP010-E-Compressor-NG middle shift tooling-1';
   ParameterElement.B2PressCylFixtureCode := 'SZ23055-OP010-E-Compressor-ring1 Upper pressing fixture-1';
   ParameterElement.R1GripperFixtureCode[0] := '';
   ParameterElement.R1GripperFixtureCode[1] := 'SZ23055-OP010-E-Compressor-robot1 ring1 Left clamping jaw tooling-1';
   ParameterElement.R1GripperFixtureCode[2] := 'SZ23055-OP010-E-Compressor-robot1 ring1 Right clamping jaw tooling-2';
   ParameterElement.R1GripperFixtureCode[3] := 'SZ23055-OP010-E-Compressor-robot1 shaft Left clamping jaw tooling-1';
   ParameterElement.R1GripperFixtureCode[4] := 'SZ23055-OP010-E-Compressor-robot1 shaft Right clamping jaw tooling-2';
   ParameterElement.R1GripperFixtureCode[5] := '';
   ParameterElement.R1GripperFixtureCode[6] := '';
   ParameterElement.R2GripperFixtureCode[0] := '';
   ParameterElement.R2GripperFixtureCode[1] := 'SZ23055-OP010-E-Compressor-robot2 shaft Right clamping jaw tooling-2';
   ParameterElement.R2GripperFixtureCode[2] := 'SZ23055-OP010-E-Compressor-robot2 shaft Left clamping jaw tooling-1';
   ParameterElement.R2GripperFixtureCode[3] := 'SZ23055-OP010-E-Compressor-robot2 magnet Left clamping jaw tooling-1';
   ParameterElement.R2GripperFixtureCode[4] := 'SZ23055-OP010-E-Compressor-robot2 magnet Right clamping jaw tooling-2';
   ParameterElement.R2GripperFixtureCode[5] := '';
   ParameterElement.R2GripperFixtureCode[6] := '';
   ParameterElement.R3GripperFixtureCode[0] := '';
   ParameterElement.R3GripperFixtureCode[1] := 'SZ23055-OP010-E-Compressor-robot3 ring2 Right clamping jaw tooling-2';
   ParameterElement.R3GripperFixtureCode[2] := 'SZ23055-OP010-E-Compressor-robot3 ring2 Left clamping jaw tooling-1';
   ParameterElement.R3GripperFixtureCode[3] := 'SZ23055-OP010-E-Compressor-robot3 shaft Left clamping jaw tooling-1';
   ParameterElement.R3GripperFixtureCode[4] := 'SZ23055-OP010-E-Compressor-robot3 shaft Right clamping jaw tooling-2';
   ParameterElement.R3GripperFixtureCode[5] := '';
   ParameterElement.R3GripperFixtureCode[6] := '';
   ParameterElement.B1PressProgram := 1;
   ParameterElement.B2PressProgram := 1;
   ParameterElement.CGlueShaftIV3Program_1 := 16#0001;
   ParameterElement.CGlueShaftIV3Program_2 := 16#0002;
   ParameterElement.CGlueShaftIV3Program_3 := 16#0003;
   ParameterElement.CGlueShaftIV3Program_4 := 16#0004;
   ParameterElement.CGlueMagnetIV3Program := 16#0001;
   ParameterElement.CGlueProgram := 1;

END_DATA_BLOCK

DATA_BLOCK "ST10_CountCycleTimeMain_DB"
{ S7_Optimized_Access := 'TRUE' }
VERSION : 0.1
NON_RETAIN
"ST10_CountCycleTimeMain"

BEGIN

END_DATA_BLOCK

DATA_BLOCK "DT-Chars_DB"
{ S7_Optimized_Access := 'FALSE' }
VERSION : 0.1
NON_RETAIN
"DT-Chars"

BEGIN

END_DATA_BLOCK

